LIN {X 0,Y 474.642,Z 379.86,A -85,B 0,C 180,E1 -7365.421,E2 -7365.421} C_VEL
LIN {X 0,Y 474.698,Z 379.855,A -85,B 0,C 180,E1 -7368.037,E2 -7368.037} C_VEL
LIN {X 0,Y 474.722,Z 379.85,A -85,B 0,C 180,E1 -7371.486,E2 -7371.486} C_VEL
LIN {X 0,Y 474.772,Z 379.846,A -85,B 0,C 180,E1 -7374.052,E2 -7374.052} C_VEL
LIN {X 0,Y 474.888,Z 379.83,A -85,B 0,C 180,E1 -7377.455,E2 -7377.455} C_VEL
LIN {X 0,Y 474.905,Z 379.83,A -85,B 0,C 180,E1 -7380,E2 -7380} C_VEL
LIN {X 0,Y 474.888,Z 379.832,A -85,B 0,C 180,E1 -7382.545,E2 -7382.545} C_VEL
LIN {X 0,Y 474.773,Z 379.846,A -85,B 0,C 180,E1 -7385.948,E2 -7385.948} C_VEL
LIN {X 0,Y 474.722,Z 379.853,A -85,B 0,C 180,E1 -7388.514,E2 -7388.514} C_VEL
LIN {X 0,Y 474.697,Z 379.856,A -85,B 0,C 180,E1 -7391.963,E2 -7391.963} C_VEL
LIN {X 0,Y 474.694,Z 379.855,A -85,B 0,C 180,E1 -7395.456,E2 -7395.456} C_VEL
LIN {X 0,Y 474.66,Z 379.858,A -85,B 0,C 180,E1 -7399.01,E2 -7399.01} C_VEL
LIN {X 0,Y 474.585,Z 379.871,A -85,B 0,C 180,E1 -7401.729,E2 -7401.729} C_VEL
LIN {X 0,Y 474.654,Z 379.86,A -85,B 0,C 180,E1 -7404.493,E2 -7404.493} C_VEL
LIN {X 0,Y 474.694,Z 379.855,A -85,B 0,C 180,E1 -7407.339,E2 -7407.339} C_VEL
LIN {X 0,Y 474.605,Z 379.865,A -85,B 0,C 180,E1 -7410.812,E2 -7410.812} C_VEL
LIN {X 0,Y 474.634,Z 379.862,A -85,B 0,C 180,E1 -7413.984,E2 -7413.984} C_VEL
LIN {X 0,Y 474.571,Z 379.869,A -85,B 0,C 180,E1 -7416.9,E2 -7416.9} C_VEL
LIN {X 0,Y 474.624,Z 379.865,A -85,B 0,C 180,E1 -7419.648,E2 -7419.648} C_VEL
LIN {X 0,Y 474.632,Z 379.862,A -85,B 0,C 180,E1 -7422.932,E2 -7422.932} C_VEL
LIN {X 0,Y 474.607,Z 379.865,A -85,B 0,C 180,E1 -7425.896,E2 -7425.896} C_VEL
LIN {X 0,Y 474.639,Z 379.862,A -85,B 0,C 180,E1 -7429.039,E2 -7429.039} C_VEL
LIN {X 0,Y 474.615,Z 379.864,A -85,B 0,C 180,E1 -7431.703,E2 -7431.703} C_VEL
LIN {X 0,Y 474.629,Z 379.861,A -85,B 0,C 180,E1 -7434.727,E2 -7434.727} C_VEL
LIN {X 0,Y 474.635,Z 379.861,A -85,B 0,C 180,E1 -7437.788,E2 -7437.788} C_VEL
LIN {X 0,Y 474.624,Z 379.864,A -85,B 0,C 180,E1 -7440.885,E2 -7440.885} C_VEL
LIN {X 0,Y 474.661,Z 379.858,A -85,B 0,C 180,E1 -7443.629,E2 -7443.629} C_VEL
LIN {X 0,Y 474.636,Z 379.861,A -85,B 0,C 180,E1 -7446.642,E2 -7446.642} C_VEL
LIN {X 0,Y 474.656,Z 379.856,A -85,B 0,C 180,E1 -7450.09,E2 -7450.09} C_VEL
LIN {X 0,Y 474.656,Z 379.857,A -85,B 0,C 180,E1 -7451.682,E2 -7451.682} C_VEL
LIN {X 0,Y 473.992,Z 379.94,A -85,B 0,C 180,E1 -7452.391,E2 -7452.391} C_VEL
LIN {X 0,Y 471.142,Z 380.3,A -85,B 0,C 180,E1 -7453.543,E2 -7453.543} C_VEL
LIN {X 0,Y 468.726,Z 380.603,A -85,B 0,C 180,E1 -7454.471,E2 -7454.471} C_VEL
LIN {X 0,Y 467.685,Z 380.731,A -85,B 0,C 180,E1 -7455.188,E2 -7455.188} C_VEL
LIN {X 0,Y 467.599,Z 380.739,A -85,B 0,C 180,E1 -7455.431,E2 -7455.431} C_VEL
LIN {X 0,Y 467.655,Z 380.734,A -85,B 0,C 180,E1 -7458.734,E2 -7458.734} C_VEL
LIN {X 0,Y 467.685,Z 380.853,A -85,B 0,C 180,E1 -7460.049,E2 -7460.049} C_VEL
LIN {X 0,Y 469.106,Z 388.705,A -85,B 0,C 180,E1 -7461.779,E2 -7461.779} C_VEL
LIN {X 0,Y 468.743,Z 398.423,A -85,B 0,C 180,E1 -7463.759,E2 -7463.759} C_VEL
LIN {X 0,Y 468.384,Z 409.921,A -85,B 0,C 180,E1 -7466.047,E2 -7466.047} C_VEL
LIN {X 0,Y 469.112,Z 414.147,A -85,B 0,C 180,E1 -7466.183,E2 -7466.183} C_VEL
LIN {X 0,Y 471.27,Z 426.346,A -85,B 0,C 180,E1 -7466.446,E2 -7466.446} C_VEL
LIN {X 0,Y 470.532,Z 517.39,A -85,B 0,C 180,E1 -7467.86,E2 -7467.86} C_VEL
LIN {X 0,Y 470.19,Z 531.181,A -85,B 0,C 180,E1 -7468.26,E2 -7468.26} C_VEL
LIN {X 0,Y 469.819,Z 544.038,A -85,B 0,C 180,E1 -7468.821,E2 -7468.821} C_VEL
LIN {X 0,Y 469.283,Z 556.55,A -85,B 0,C 180,E1 -7469.571,E2 -7469.571} C_VEL
LIN {X 0,Y 468.732,Z 567.702,A -85,B 0,C 180,E1 -7470.429,E2 -7470.429} C_VEL
LIN {X 0,Y 468.308,Z 576.724,A -85,B 0,C 180,E1 -7471.29,E2 -7471.29} C_VEL
LIN {X 0,Y 467.868,Z 586.01,A -85,B 0,C 180,E1 -7472.367,E2 -7472.367} C_VEL
LIN {X 0,Y 467.406,Z 595.008,A -85,B 0,C 180,E1 -7473.664,E2 -7473.664} C_VEL
LIN {X 0,Y 467.034,Z 602.282,A -85,B 0,C 180,E1 -7474.964,E2 -7474.964} C_VEL
LIN {X 0,Y 466.932,Z 608.355,A -85,B 0,C 180,E1 -7476.328,E2 -7476.328} C_VEL
LIN {X 0,Y 466.768,Z 613.344,A -85,B 0,C 180,E1 -7477.788,E2 -7477.788} C_VEL
LIN {X 0,Y 466.684,Z 615.684,A -85,B 0,C 180,E1 -7478.661,E2 -7478.661} C_VEL
LIN {X 0,Y 466.575,Z 617.597,A -85,B 0,C 180,E1 -7479.537,E2 -7479.537} C_VEL
LIN {X 0,Y 466.601,Z 619.039,A -85,B 0,C 180,E1 -7480.413,E2 -7480.413} C_VEL
LIN {X 0,Y 466.627,Z 620.462,A -85,B 0,C 180,E1 -7481.767,E2 -7481.767} C_VEL
LIN {X 0,Y 466.545,Z 620.916,A -85,B 0,C 180,E1 -7483.059,E2 -7483.059} C_VEL
LIN {X 0,Y 466.506,Z 620.687,A -85,B 0,C 180,E1 -7483.948,E2 -7483.948} C_VEL
LIN {X 0,Y 466.582,Z 619.413,A -85,B 0,C 180,E1 -7485.417,E2 -7485.417} C_VEL
LIN {X 0,Y 466.575,Z 617.498,A -85,B 0,C 180,E1 -7486.63,E2 -7486.63} C_VEL
LIN {X 0,Y 466.722,Z 614.362,A -85,B 0,C 180,E1 -7487.98,E2 -7487.98} C_VEL
LIN {X 0,Y 466.873,Z 610.064,A -85,B 0,C 180,E1 -7489.339,E2 -7489.339} C_VEL
LIN {X 0,Y 467.114,Z 603.53,A -85,B 0,C 180,E1 -7490.908,E2 -7490.908} C_VEL
LIN {X 0,Y 467.476,Z 596.001,A -85,B 0,C 180,E1 -7492.309,E2 -7492.309} C_VEL
LIN {X 0,Y 467.885,Z 587.185,A -85,B 0,C 180,E1 -7493.613,E2 -7493.613} C_VEL
LIN {X 0,Y 468.357,Z 577.917,A -85,B 0,C 180,E1 -7494.725,E2 -7494.725} C_VEL
LIN {X 0,Y 468.885,Z 567.133,A -85,B 0,C 180,E1 -7495.764,E2 -7495.764} C_VEL
LIN {X 0,Y 469.394,Z 556.525,A -85,B 0,C 180,E1 -7496.58,E2 -7496.58} C_VEL
LIN {X 0,Y 469.876,Z 545.344,A -85,B 0,C 180,E1 -7497.261,E2 -7497.261} C_VEL
LIN {X 0,Y 470.301,Z 533.471,A -85,B 0,C 180,E1 -7497.81,E2 -7497.81} C_VEL
LIN {X 0,Y 470.598,Z 520.548,A -85,B 0,C 180,E1 -7498.222,E2 -7498.222} C_VEL
LIN {X 0,Y 470.832,Z 503.541,A -85,B 0,C 180,E1 -7498.532,E2 -7498.532} C_VEL
LIN {X 0,Y 471.437,Z 425.884,A -85,B 0,C 180,E1 -7499.73,E2 -7499.73} C_VEL
LIN {X 0,Y 468.522,Z 410.206,A -85,B 0,C 180,E1 -7500.122,E2 -7500.122} C_VEL
LIN {X 0,Y 468.767,Z 404.216,A -85,B 0,C 180,E1 -7501.287,E2 -7501.287} C_VEL
LIN {X 0,Y 469.373,Z 391.54,A -85,B 0,C 180,E1 -7503.899,E2 -7503.899} C_VEL
LIN {X 0,Y 468.511,Z 385.277,A -85,B 0,C 180,E1 -7505.276,E2 -7505.276} C_VEL
LIN {X 0,Y 467.577,Z 380.785,A -85,B 0,C 180,E1 -7506.353,E2 -7506.353} C_VEL
LIN {X 0,Y 467.615,Z 380.739,A -85,B 0,C 180,E1 -7509.14,E2 -7509.14} C_VEL
LIN {X 0,Y 467.615,Z 380.737,A -85,B 0,C 180,E1 -7512.571,E2 -7512.571} C_VEL
LIN {X 0,Y 467.569,Z 380.74,A -85,B 0,C 180,E1 -7516.176,E2 -7516.176} C_VEL
LIN {X 0,Y 467.585,Z 380.737,A -85,B 0,C 180,E1 -7518.721,E2 -7518.721} C_VEL
LIN {X 0,Y 467.572,Z 380.739,A -85,B 0,C 180,E1 -7521.406,E2 -7521.406} C_VEL
LIN {X 0,Y 467.557,Z 380.74,A -85,B 0,C 180,E1 -7524.259,E2 -7524.259} C_VEL
LIN {X 0,Y 467.575,Z 380.743,A -85,B 0,C 180,E1 -7527.32,E2 -7527.32} C_VEL
LIN {X 0,Y 467.571,Z 380.732,A -85,B 0,C 180,E1 -7530.665,E2 -7530.665} C_VEL
LIN {X 0,Y 467.62,Z 380.738,A -85,B 0,C 180,E1 -7533.2,E2 -7533.2} C_VEL
LIN {X 0,Y 467.585,Z 380.739,A -85,B 0,C 180,E1 -7536.467,E2 -7536.467} C_VEL
LIN {X 0,Y 467.617,Z 380.733,A -85,B 0,C 180,E1 -7539.777,E2 -7539.777} C_VEL
LIN {X 0,Y 467.6,Z 380.735,A -85,B 0,C 180,E1 -7542.506,E2 -7542.506} C_VEL
LIN {X 0,Y 467.598,Z 380.736,A -85,B 0,C 180,E1 -7545.196,E2 -7545.196} C_VEL
LIN {X 0,Y 467.673,Z 380.726,A -85,B 0,C 180,E1 -7547.855,E2 -7547.855} C_VEL
LIN {X 0,Y 467.674,Z 380.728,A -85,B 0,C 180,E1 -7551.357,E2 -7551.357} C_VEL
LIN {X 0,Y 467.738,Z 380.714,A -85,B 0,C 180,E1 -7553.963,E2 -7553.963} C_VEL
LIN {X 0,Y 467.858,Z 380.703,A -85,B 0,C 180,E1 -7557.417,E2 -7557.417} C_VEL
LIN {X 0,Y 467.873,Z 380.698,A -85,B 0,C 180,E1 -7560,E2 -7560} C_VEL
LIN {X 0,Y 467.852,Z 380.709,A -85,B 0,C 180,E1 -7562.583,E2 -7562.583} C_VEL
LIN {X 0,Y 467.739,Z 380.718,A -85,B 0,C 180,E1 -7566.038,E2 -7566.038} C_VEL
LIN {X 0,Y 467.674,Z 380.727,A -85,B 0,C 180,E1 -7568.643,E2 -7568.643} C_VEL
LIN {X 0,Y 467.674,Z 380.727,A -85,B 0,C 180,E1 -7572.145,E2 -7572.145} C_VEL
LIN {X 0,Y 467.64,Z 380.73,A -85,B 0,C 180,E1 -7575.886,E2 -7575.886} C_VEL
LIN {X 0,Y 467.616,Z 380.733,A -85,B 0,C 180,E1 -7579.308,E2 -7579.308} C_VEL
LIN {X 0,Y 467.534,Z 380.743,A -85,B 0,C 180,E1 -7582.074,E2 -7582.074} C_VEL
LIN {X 0,Y 467.598,Z 380.739,A -85,B 0,C 180,E1 -7584.888,E2 -7584.888} C_VEL
LIN {X 0,Y 467.62,Z 380.731,A -85,B 0,C 180,E1 -7587.769,E2 -7587.769} C_VEL
LIN {X 0,Y 467.562,Z 380.742,A -85,B 0,C 180,E1 -7591.046,E2 -7591.046} C_VEL
LIN {X 0,Y 467.584,Z 380.739,A -85,B 0,C 180,E1 -7594.243,E2 -7594.243} C_VEL
LIN {X 0,Y 467.545,Z 380.741,A -85,B 0,C 180,E1 -7597.188,E2 -7597.188} C_VEL
LIN {X 0,Y 467.591,Z 380.74,A -85,B 0,C 180,E1 -7600.263,E2 -7600.263} C_VEL
LIN {X 0,Y 467.614,Z 380.732,A -85,B 0,C 180,E1 -7602.572,E2 -7602.572} C_VEL
LIN {X 0,Y 467.563,Z 380.739,A -85,B 0,C 180,E1 -7606.178,E2 -7606.178} C_VEL
LIN {X 0,Y 467.578,Z 380.741,A -85,B 0,C 180,E1 -7608.724,E2 -7608.724} C_VEL
LIN {X 0,Y 467.564,Z 380.743,A -85,B 0,C 180,E1 -7611.957,E2 -7611.957} C_VEL
LIN {X 0,Y 467.567,Z 380.74,A -85,B 0,C 180,E1 -7615.169,E2 -7615.169} C_VEL
LIN {X 0,Y 467.583,Z 380.741,A -85,B 0,C 180,E1 -7618.261,E2 -7618.261} C_VEL
LIN {X 0,Y 467.577,Z 380.741,A -85,B 0,C 180,E1 -7621.251,E2 -7621.251} C_VEL
LIN {X 0,Y 467.612,Z 380.739,A -85,B 0,C 180,E1 -7624.161,E2 -7624.161} C_VEL
LIN {X 0,Y 467.657,Z 380.901,A -85,B 0,C 180,E1 -7624.903,E2 -7624.903} C_VEL
LIN {X 0,Y 469.631,Z 391.304,A -85,B 0,C 180,E1 -7627.103,E2 -7627.103} C_VEL
LIN {X 0,Y 469.655,Z 396.068,A -85,B 0,C 180,E1 -7628.032,E2 -7628.032} C_VEL
LIN {X 0,Y 468.787,Z 414.077,A -85,B 0,C 180,E1 -7631.438,E2 -7631.438} C_VEL
LIN {X 0,Y 468.449,Z 422.17,A -85,B 0,C 180,E1 -7632.905,E2 -7632.905} C_VEL
LIN {X 0,Y 469.901,Z 430.791,A -85,B 0,C 180,E1 -7633.133,E2 -7633.133} C_VEL
LIN {X 0,Y 471.376,Z 440.03,A -85,B 0,C 180,E1 -7633.338,E2 -7633.338} C_VEL
LIN {X 0,Y 470.646,Z 529.828,A -85,B 0,C 180,E1 -7634.741,E2 -7634.741} C_VEL
LIN {X 0,Y 470.312,Z 543.065,A -85,B 0,C 180,E1 -7635.118,E2 -7635.118} C_VEL
LIN {X 0,Y 469.856,Z 555.767,A -85,B 0,C 180,E1 -7635.657,E2 -7635.657} C_VEL
LIN {X 0,Y 469.352,Z 567.861,A -85,B 0,C 180,E1 -7636.36,E2 -7636.36} C_VEL
LIN {X 0,Y 468.852,Z 578.48,A -85,B 0,C 180,E1 -7637.152,E2 -7637.152} C_VEL
LIN {X 0,Y 468.356,Z 589.73,A -85,B 0,C 180,E1 -7638.203,E2 -7638.203} C_VEL
LIN {X 0,Y 467.884,Z 598.212,A -85,B 0,C 180,E1 -7639.178,E2 -7639.178} C_VEL
LIN {X 0,Y 467.442,Z 607.416,A -85,B 0,C 180,E1 -7640.481,E2 -7640.481} C_VEL
LIN {X 0,Y 467.118,Z 614.819,A -85,B 0,C 180,E1 -7641.783,E2 -7641.783} C_VEL
LIN {X 0,Y 466.912,Z 620.766,A -85,B 0,C 180,E1 -7643.084,E2 -7643.084} C_VEL
LIN {X 0,Y 466.794,Z 625.466,A -85,B 0,C 180,E1 -7644.384,E2 -7644.384} C_VEL
LIN {X 0,Y 466.648,Z 629.056,A -85,B 0,C 180,E1 -7645.682,E2 -7645.682} C_VEL
LIN {X 0,Y 466.661,Z 630.908,A -85,B 0,C 180,E1 -7646.547,E2 -7646.547} C_VEL
LIN {X 0,Y 466.644,Z 632.297,A -85,B 0,C 180,E1 -7647.411,E2 -7647.411} C_VEL
LIN {X 0,Y 466.589,Z 633.893,A -85,B 0,C 180,E1 -7649.137,E2 -7649.137} C_VEL
LIN {X 0,Y 466.598,Z 634.105,A -85,B 0,C 180,E1 -7650,E2 -7650} C_VEL
LIN {X 0,Y 466.604,Z 633.278,A -85,B 0,C 180,E1 -7651.726,E2 -7651.726} C_VEL
LIN {X 0,Y 466.644,Z 632.283,A -85,B 0,C 180,E1 -7652.59,E2 -7652.59} C_VEL
LIN {X 0,Y 466.661,Z 630.885,A -85,B 0,C 180,E1 -7653.454,E2 -7653.454} C_VEL
LIN {X 0,Y 466.693,Z 627.949,A -85,B 0,C 180,E1 -7654.751,E2 -7654.751} C_VEL
LIN {X 0,Y 466.784,Z 623.972,A -85,B 0,C 180,E1 -7656.05,E2 -7656.05} C_VEL
LIN {X 0,Y 466.982,Z 617.847,A -85,B 0,C 180,E1 -7657.567,E2 -7657.567} C_VEL
LIN {X 0,Y 467.303,Z 611.156,A -85,B 0,C 180,E1 -7658.868,E2 -7658.868} C_VEL
LIN {X 0,Y 467.63,Z 602.848,A -85,B 0,C 180,E1 -7660.171,E2 -7660.171} C_VEL
LIN {X 0,Y 468.078,Z 594.311,A -85,B 0,C 180,E1 -7661.256,E2 -7661.256} C_VEL
LIN {X 0,Y 468.605,Z 583.971,A -85,B 0,C 180,E1 -7662.321,E2 -7662.321} C_VEL
LIN {X 0,Y 469.029,Z 573.591,A -85,B 0,C 180,E1 -7663.187,E2 -7663.187} C_VEL
LIN {X 0,Y 469.49,Z 561.79,A -85,B 0,C 180,E1 -7663.968,E2 -7663.968} C_VEL
LIN {X 0,Y 469.979,Z 549.854,A -85,B 0,C 180,E1 -7664.561,E2 -7664.561} C_VEL
LIN {X 0,Y 470.373,Z 536.957,A -85,B 0,C 180,E1 -7665.019,E2 -7665.019} C_VEL
LIN {X 0,Y 470.588,Z 523.354,A -85,B 0,C 180,E1 -7665.317,E2 -7665.317} C_VEL
LIN {X 0,Y 471.188,Z 439.488,A -85,B 0,C 180,E1 -7666.6,E2 -7666.6} C_VEL
LIN {X 0,Y 468.374,Z 422.324,A -85,B 0,C 180,E1 -7666.986,E2 -7666.986} C_VEL
LIN {X 0,Y 468.713,Z 413.473,A -85,B 0,C 180,E1 -7668.565,E2 -7668.565} C_VEL
LIN {X 0,Y 469.571,Z 393.96,A -85,B 0,C 180,E1 -7672.204,E2 -7672.204} C_VEL
LIN {X 0,Y 469.415,Z 390.298,A -85,B 0,C 180,E1 -7672.909,E2 -7672.909} C_VEL
LIN {X 0,Y 467.723,Z 381.106,A -85,B 0,C 180,E1 -7674.762,E2 -7674.762} C_VEL
LIN {X 0,Y 467.626,Z 380.739,A -85,B 0,C 180,E1 -7675.099,E2 -7675.099} C_VEL
LIN {X 0,Y 467.628,Z 380.736,A -85,B 0,C 180,E1 -7677.768,E2 -7677.768} C_VEL
LIN {X 0,Y 467.57,Z 380.743,A -85,B 0,C 180,E1 -7681.045,E2 -7681.045} C_VEL
LIN {X 0,Y 467.59,Z 380.737,A -85,B 0,C 180,E1 -7684.242,E2 -7684.242} C_VEL
LIN {X 0,Y 467.552,Z 380.745,A -85,B 0,C 180,E1 -7687.186,E2 -7687.186} C_VEL
LIN {X 0,Y 467.578,Z 380.738,A -85,B 0,C 180,E1 -7690.264,E2 -7690.264} C_VEL
LIN {X 0,Y 467.585,Z 380.738,A -85,B 0,C 180,E1 -7692.566,E2 -7692.566} C_VEL
LIN {X 0,Y 467.569,Z 380.743,A -85,B 0,C 180,E1 -7695.053,E2 -7695.053} C_VEL
LIN {X 0,Y 467.622,Z 380.738,A -85,B 0,C 180,E1 -7697.443,E2 -7697.443} C_VEL
LIN {X 0,Y 467.616,Z 380.736,A -85,B 0,C 180,E1 -7700.858,E2 -7700.858} C_VEL
LIN {X 0,Y 467.56,Z 380.742,A -85,B 0,C 180,E1 -7704.26,E2 -7704.26} C_VEL
LIN {X 0,Y 467.578,Z 380.743,A -85,B 0,C 180,E1 -7707.32,E2 -7707.32} C_VEL
LIN {X 0,Y 467.566,Z 380.742,A -85,B 0,C 180,E1 -7710.667,E2 -7710.667} C_VEL
LIN {X 0,Y 467.623,Z 380.738,A -85,B 0,C 180,E1 -7713.2,E2 -7713.2} C_VEL
LIN {X 0,Y 467.588,Z 380.74,A -85,B 0,C 180,E1 -7716.468,E2 -7716.468} C_VEL
LIN {X 0,Y 467.619,Z 380.735,A -85,B 0,C 180,E1 -7719.777,E2 -7719.777} C_VEL
LIN {X 0,Y 467.604,Z 380.738,A -85,B 0,C 180,E1 -7722.506,E2 -7722.506} C_VEL
LIN {X 0,Y 467.6,Z 380.739,A -85,B 0,C 180,E1 -7725.196,E2 -7725.196} C_VEL
LIN {X 0,Y 467.649,Z 380.732,A -85,B 0,C 180,E1 -7727.854,E2 -7727.854} C_VEL
LIN {X 0,Y 467.675,Z 380.728,A -85,B 0,C 180,E1 -7731.357,E2 -7731.357} C_VEL
LIN {X 0,Y 467.737,Z 380.722,A -85,B 0,C 180,E1 -7733.962,E2 -7733.962} C_VEL
LIN {X 0,Y 467.854,Z 380.706,A -85,B 0,C 180,E1 -7737.417,E2 -7737.417} C_VEL
LIN {X 0,Y 467.876,Z 380.705,A -85,B 0,C 180,E1 -7740,E2 -7740} C_VEL
LIN {X 0,Y 467.854,Z 380.708,A -85,B 0,C 180,E1 -7742.583,E2 -7742.583} C_VEL
LIN {X 0,Y 467.737,Z 380.722,A -85,B 0,C 180,E1 -7746.037,E2 -7746.037} C_VEL
LIN {X 0,Y 467.675,Z 380.731,A -85,B 0,C 180,E1 -7748.643,E2 -7748.643} C_VEL
LIN {X 0,Y 467.649,Z 380.733,A -85,B 0,C 180,E1 -7752.146,E2 -7752.146} C_VEL
LIN {X 0,Y 467.633,Z 380.737,A -85,B 0,C 180,E1 -7755.695,E2 -7755.695} C_VEL
LIN {X 0,Y 467.612,Z 380.737,A -85,B 0,C 180,E1 -7758.765,E2 -7758.765} C_VEL
LIN {X 0,Y 467.575,Z 380.741,A -85,B 0,C 180,E1 -7761.269,E2 -7761.269} C_VEL
LIN {X 0,Y 467.568,Z 380.743,A -85,B 0,C 180,E1 -7763.944,E2 -7763.944} C_VEL
LIN {X 0,Y 467.622,Z 380.735,A -85,B 0,C 180,E1 -7766.8,E2 -7766.8} C_VEL
LIN {X 0,Y 467.583,Z 380.742,A -85,B 0,C 180,E1 -7769.736,E2 -7769.736} C_VEL
LIN {X 0,Y 467.579,Z 380.74,A -85,B 0,C 180,E1 -7772.759,E2 -7772.759} C_VEL
LIN {X 0,Y 467.553,Z 380.744,A -85,B 0,C 180,E1 -7775.89,E2 -7775.89} C_VEL
LIN {X 0,Y 467.579,Z 380.742,A -85,B 0,C 180,E1 -7779.145,E2 -7779.145} C_VEL
LIN {X 0,Y 467.583,Z 380.739,A -85,B 0,C 180,E1 -7782.567,E2 -7782.567} C_VEL
LIN {X 0,Y 467.568,Z 380.743,A -85,B 0,C 180,E1 -7785.054,E2 -7785.054} C_VEL
LIN {X 0,Y 467.586,Z 380.742,A -85,B 0,C 180,E1 -7787.44,E2 -7787.44} C_VEL
LIN {X 0,Y 467.614,Z 380.736,A -85,B 0,C 180,E1 -7790.859,E2 -7790.859} C_VEL
LIN {X 0,Y 467.562,Z 380.741,A -85,B 0,C 180,E1 -7794.261,E2 -7794.261} C_VEL
LIN {X 0,Y 467.581,Z 380.743,A -85,B 0,C 180,E1 -7797.321,E2 -7797.321} C_VEL
LIN {X 0,Y 467.57,Z 380.741,A -85,B 0,C 180,E1 -7800.668,E2 -7800.668} C_VEL
LIN {X 0,Y 467.617,Z 380.739,A -85,B 0,C 180,E1 -7803.2,E2 -7803.2} C_VEL
LIN {X 0,Y 467.593,Z 380.737,A -85,B 0,C 180,E1 -7806.469,E2 -7806.469} C_VEL
LIN {X 0,Y 467.624,Z 380.733,A -85,B 0,C 180,E1 -7809.777,E2 -7809.777} C_VEL
LIN {X 0,Y 467.608,Z 380.736,A -85,B 0,C 180,E1 -7812.507,E2 -7812.507} C_VEL
LIN {X 0,Y 467.599,Z 380.739,A -85,B 0,C 180,E1 -7815.431,E2 -7815.431} C_VEL
LIN {X 0,Y 466.928,Z 380.82,A -85,B 0,C 180,E1 -7816.15,E2 -7816.15} C_VEL
LIN {X 0,Y 464.085,Z 381.178,A -85,B 0,C 180,E1 -7817.319,E2 -7817.319} C_VEL
LIN {X 0,Y 461.686,Z 381.476,A -85,B 0,C 180,E1 -7818.261,E2 -7818.261} C_VEL
LIN {X 0,Y 460.66,Z 381.605,A -85,B 0,C 180,E1 -7818.988,E2 -7818.988} C_VEL
LIN {X 0,Y 460.579,Z 381.614,A -85,B 0,C 180,E1 -7819.235,E2 -7819.235} C_VEL
LIN {X 0,Y 460.657,Z 381.768,A -85,B 0,C 180,E1 -7819.895,E2 -7819.895} C_VEL
LIN {X 0,Y 462.108,Z 389.84,A -85,B 0,C 180,E1 -7821.691,E2 -7821.691} C_VEL
LIN {X 0,Y 461.936,Z 398.299,A -85,B 0,C 180,E1 -7823.448,E2 -7823.448} C_VEL
LIN {X 0,Y 461.698,Z 401.507,A -85,B 0,C 180,E1 -7824.102,E2 -7824.102} C_VEL
LIN {X 0,Y 461.395,Z 409.977,A -85,B 0,C 180,E1 -7825.796,E2 -7825.796} C_VEL
LIN {X 0,Y 461.901,Z 412.882,A -85,B 0,C 180,E1 -7825.91,E2 -7825.91} C_VEL
LIN {X 0,Y 464.4,Z 425.885,A -85,B 0,C 180,E1 -7826.204,E2 -7826.204} C_VEL
LIN {X 0,Y 463.665,Z 517.07,A -85,B 0,C 180,E1 -7827.638,E2 -7827.638} C_VEL
LIN {X 0,Y 463.326,Z 530.256,A -85,B 0,C 180,E1 -7828.017,E2 -7828.017} C_VEL
LIN {X 0,Y 462.916,Z 543.441,A -85,B 0,C 180,E1 -7828.586,E2 -7828.586} C_VEL
LIN {X 0,Y 462.456,Z 554.555,A -85,B 0,C 180,E1 -7829.238,E2 -7829.238} C_VEL
LIN {X 0,Y 461.879,Z 566.094,A -85,B 0,C 180,E1 -7830.109,E2 -7830.109} C_VEL
LIN {X 0,Y 461.329,Z 576.484,A -85,B 0,C 180,E1 -7831.091,E2 -7831.091} C_VEL
LIN {X 0,Y 460.871,Z 585.849,A -85,B 0,C 180,E1 -7832.185,E2 -7832.185} C_VEL
LIN {X 0,Y 460.373,Z 594.9,A -85,B 0,C 180,E1 -7833.501,E2 -7833.501} C_VEL
LIN {X 0,Y 459.994,Z 602.211,A -85,B 0,C 180,E1 -7834.82,E2 -7834.82} C_VEL
LIN {X 0,Y 459.89,Z 608.063,A -85,B 0,C 180,E1 -7836.141,E2 -7836.141} C_VEL
LIN {X 0,Y 459.697,Z 612.705,A -85,B 0,C 180,E1 -7837.466,E2 -7837.466} C_VEL
LIN {X 0,Y 459.565,Z 616.245,A -85,B 0,C 180,E1 -7838.796,E2 -7838.796} C_VEL
LIN {X 0,Y 459.475,Z 618.035,A -85,B 0,C 180,E1 -7839.686,E2 -7839.686} C_VEL
LIN {X 0,Y 459.497,Z 619.384,A -85,B 0,C 180,E1 -7840.576,E2 -7840.576} C_VEL
LIN {X 0,Y 459.546,Z 620.598,A -85,B 0,C 180,E1 -7841.826,E2 -7841.826} C_VEL
LIN {X 0,Y 459.428,Z 620.987,A -85,B 0,C 180,E1 -7843.265,E2 -7843.265} C_VEL
LIN {X 0,Y 459.43,Z 620.682,A -85,B 0,C 180,E1 -7844.167,E2 -7844.167} C_VEL
LIN {X 0,Y 459.493,Z 619.461,A -85,B 0,C 180,E1 -7845.508,E2 -7845.508} C_VEL
LIN {X 0,Y 459.558,Z 616.248,A -85,B 0,C 180,E1 -7847.35,E2 -7847.35} C_VEL
LIN {X 0,Y 459.728,Z 612.577,A -85,B 0,C 180,E1 -7848.725,E2 -7848.725} C_VEL
LIN {X 0,Y 459.895,Z 607.676,A -85,B 0,C 180,E1 -7850.11,E2 -7850.11} C_VEL
LIN {X 0,Y 460.171,Z 601.386,A -85,B 0,C 180,E1 -7851.502,E2 -7851.502} C_VEL
LIN {X 0,Y 460.594,Z 593.467,A -85,B 0,C 180,E1 -7852.897,E2 -7852.897} C_VEL
LIN {X 0,Y 461.085,Z 584.547,A -85,B 0,C 180,E1 -7854.149,E2 -7854.149} C_VEL
LIN {X 0,Y 461.536,Z 575.027,A -85,B 0,C 180,E1 -7855.236,E2 -7855.236} C_VEL
LIN {X 0,Y 462.166,Z 563.828,A -85,B 0,C 180,E1 -7856.265,E2 -7856.265} C_VEL
LIN {X 0,Y 462.664,Z 552.064,A -85,B 0,C 180,E1 -7857.11,E2 -7857.11} C_VEL
LIN {X 0,Y 463.289,Z 539.303,A -85,B 0,C 180,E1 -7857.805,E2 -7857.805} C_VEL
LIN {X 0,Y 463.668,Z 526.393,A -85,B 0,C 180,E1 -7858.306,E2 -7858.306} C_VEL
LIN {X 0,Y 463.927,Z 512.622,A -85,B 0,C 180,E1 -7858.641,E2 -7858.641} C_VEL
LIN {X 0,Y 464.605,Z 426.038,A -85,B 0,C 180,E1 -7860.009,E2 -7860.009} C_VEL
LIN {X 0,Y 461.61,Z 410.294,A -85,B 0,C 180,E1 -7860.419,E2 -7860.419} C_VEL
LIN {X 0,Y 461.732,Z 406.389,A -85,B 0,C 180,E1 -7861.165,E2 -7861.165} C_VEL
LIN {X 0,Y 462.432,Z 393.06,A -85,B 0,C 180,E1 -7863.952,E2 -7863.952} C_VEL
LIN {X 0,Y 461.896,Z 388.331,A -85,B 0,C 180,E1 -7865.001,E2 -7865.001} C_VEL
LIN {X 0,Y 460.519,Z 381.649,A -85,B 0,C 180,E1 -7866.609,E2 -7866.609} C_VEL
LIN {X 0,Y 460.575,Z 381.615,A -85,B 0,C 180,E1 -7869.857,E2 -7869.857} C_VEL
LIN {X 0,Y 460.538,Z 381.618,A -85,B 0,C 180,E1 -7872.904,E2 -7872.904} C_VEL
LIN {X 0,Y 460.519,Z 381.619,A -85,B 0,C 180,E1 -7875.828,E2 -7875.828} C_VEL
LIN {X 0,Y 460.538,Z 381.618,A -85,B 0,C 180,E1 -7878.989,E2 -7878.989} C_VEL
LIN {X 0,Y 460.541,Z 381.614,A -85,B 0,C 180,E1 -7881.268,E2 -7881.268} C_VEL
LIN {X 0,Y 460.507,Z 381.62,A -85,B 0,C 180,E1 -7884.554,E2 -7884.554} C_VEL
LIN {X 0,Y 460.526,Z 381.618,A -85,B 0,C 180,E1 -7887.715,E2 -7887.715} C_VEL
LIN {X 0,Y 460.54,Z 381.609,A -85,B 0,C 180,E1 -7890.769,E2 -7890.769} C_VEL
LIN {X 0,Y 460.56,Z 381.612,A -85,B 0,C 180,E1 -7893.735,E2 -7893.735} C_VEL
LIN {X 0,Y 460.539,Z 381.619,A -85,B 0,C 180,E1 -7896.624,E2 -7896.624} C_VEL
LIN {X 0,Y 460.563,Z 381.614,A -85,B 0,C 180,E1 -7899.453,E2 -7899.453} C_VEL
LIN {X 0,Y 460.55,Z 381.611,A -85,B 0,C 180,E1 -7902.23,E2 -7902.23} C_VEL
LIN {X 0,Y 460.556,Z 381.615,A -85,B 0,C 180,E1 -7904.965,E2 -7904.965} C_VEL
LIN {X 0,Y 460.619,Z 381.605,A -85,B 0,C 180,E1 -7907.666,E2 -7907.666} C_VEL
LIN {X 0,Y 460.621,Z 381.608,A -85,B 0,C 180,E1 -7911.224,E2 -7911.224} C_VEL
LIN {X 0,Y 460.704,Z 381.59,A -85,B 0,C 180,E1 -7913.87,E2 -7913.87} C_VEL
LIN {X 0,Y 460.824,Z 381.579,A -85,B 0,C 180,E1 -7917.378,E2 -7917.378} C_VEL
LIN {X 0,Y 460.844,Z 381.574,A -85,B 0,C 180,E1 -7920,E2 -7920} C_VEL
LIN {X 0,Y 460.817,Z 381.585,A -85,B 0,C 180,E1 -7922.622,E2 -7922.622} C_VEL
LIN {X 0,Y 460.704,Z 381.594,A -85,B 0,C 180,E1 -7926.13,E2 -7926.13} C_VEL
LIN {X 0,Y 460.621,Z 381.605,A -85,B 0,C 180,E1 -7928.776,E2 -7928.776} C_VEL
LIN {X 0,Y 460.625,Z 381.608,A -85,B 0,C 180,E1 -7932.457,E2 -7932.457} C_VEL
LIN {X 0,Y 460.591,Z 381.609,A -85,B 0,C 180,E1 -7935.998,E2 -7935.998} C_VEL
LIN {X 0,Y 460.562,Z 381.615,A -85,B 0,C 180,E1 -7938.902,E2 -7938.902} C_VEL
LIN {X 0,Y 460.51,Z 381.617,A -85,B 0,C 180,E1 -7941.486,E2 -7941.486} C_VEL
LIN {X 0,Y 460.536,Z 381.617,A -85,B 0,C 180,E1 -7944.333,E2 -7944.333} C_VEL
LIN {X 0,Y 460.576,Z 381.61,A -85,B 0,C 180,E1 -7947.244,E2 -7947.244} C_VEL
LIN {X 0,Y 460.504,Z 381.621,A -85,B 0,C 180,E1 -7950.241,E2 -7950.241} C_VEL
LIN {X 0,Y 460.523,Z 381.616,A -85,B 0,C 180,E1 -7953.326,E2 -7953.326} C_VEL
LIN {X 0,Y 460.473,Z 381.629,A -85,B 0,C 180,E1 -7956.53,E2 -7956.53} C_VEL
LIN {X 0,Y 460.571,Z 381.611,A -85,B 0,C 180,E1 -7959.859,E2 -7959.859} C_VEL
LIN {X 0,Y 460.539,Z 381.618,A -85,B 0,C 180,E1 -7962.905,E2 -7962.905} C_VEL
LIN {X 0,Y 460.515,Z 381.615,A -85,B 0,C 180,E1 -7965.83,E2 -7965.83} C_VEL
LIN {X 0,Y 460.53,Z 381.616,A -85,B 0,C 180,E1 -7968.99,E2 -7968.99} C_VEL
LIN {X 0,Y 460.524,Z 381.618,A -85,B 0,C 180,E1 -7971.268,E2 -7971.268} C_VEL
LIN {X 0,Y 460.512,Z 381.624,A -85,B 0,C 180,E1 -7974.556,E2 -7974.556} C_VEL
LIN {X 0,Y 460.531,Z 381.618,A -85,B 0,C 180,E1 -7977.717,E2 -7977.717} C_VEL
LIN {X 0,Y 460.54,Z 381.621,A -85,B 0,C 180,E1 -7980.77,E2 -7980.77} C_VEL
LIN {X 0,Y 460.568,Z 381.617,A -85,B 0,C 180,E1 -7983.736,E2 -7983.736} C_VEL
LIN {X 0,Y 460.632,Z 381.838,A -85,B 0,C 180,E1 -7984.67,E2 -7984.67} C_VEL
LIN {X 0,Y 462.686,Z 392.573,A -85,B 0,C 180,E1 -7986.976,E2 -7986.976} C_VEL
LIN {X 0,Y 462.739,Z 397.174,A -85,B 0,C 180,E1 -7987.89,E2 -7987.89} C_VEL
LIN {X 0,Y 461.8,Z 415.227,A -85,B 0,C 180,E1 -7991.362,E2 -7991.362} C_VEL
LIN {X 0,Y 461.486,Z 421.95,A -85,B 0,C 180,E1 -7992.607,E2 -7992.607} C_VEL
LIN {X 0,Y 462.785,Z 429.059,A -85,B 0,C 180,E1 -7992.811,E2 -7992.811} C_VEL
LIN {X 0,Y 464.656,Z 441.523,A -85,B 0,C 180,E1 -7993.09,E2 -7993.09} C_VEL
LIN {X 0,Y 463.833,Z 530.506,A -85,B 0,C 180,E1 -7994.512,E2 -7994.512} C_VEL
LIN {X 0,Y 463.426,Z 544.235,A -85,B 0,C 180,E1 -7994.92,E2 -7994.92} C_VEL
LIN {X 0,Y 462.958,Z 557.078,A -85,B 0,C 180,E1 -7995.495,E2 -7995.495} C_VEL
LIN {X 0,Y 462.452,Z 568.322,A -85,B 0,C 180,E1 -7996.174,E2 -7996.174} C_VEL
LIN {X 0,Y 461.88,Z 579.389,A -85,B 0,C 180,E1 -7997.025,E2 -7997.025} C_VEL
LIN {X 0,Y 461.396,Z 589.784,A -85,B 0,C 180,E1 -7998.022,E2 -7998.022} C_VEL
LIN {X 0,Y 460.896,Z 598.234,A -85,B 0,C 180,E1 -7999.012,E2 -7999.012} C_VEL
LIN {X 0,Y 460.412,Z 607.403,A -85,B 0,C 180,E1 -8000.334,E2 -8000.334} C_VEL
LIN {X 0,Y 460.077,Z 614.787,A -85,B 0,C 180,E1 -8001.656,E2 -8001.656} C_VEL
LIN {X 0,Y 459.846,Z 620.718,A -85,B 0,C 180,E1 -8002.977,E2 -8002.977} C_VEL
LIN {X 0,Y 459.712,Z 625.405,A -85,B 0,C 180,E1 -8004.297,E2 -8004.297} C_VEL
LIN {X 0,Y 459.566,Z 628.984,A -85,B 0,C 180,E1 -8005.615,E2 -8005.615} C_VEL
LIN {X 0,Y 459.558,Z 630.828,A -85,B 0,C 180,E1 -8006.493,E2 -8006.493} C_VEL
LIN {X 0,Y 459.566,Z 632.21,A -85,B 0,C 180,E1 -8007.371,E2 -8007.371} C_VEL
LIN {X 0,Y 459.494,Z 633.798,A -85,B 0,C 180,E1 -8009.124,E2 -8009.124} C_VEL
LIN {X 0,Y 459.501,Z 634.004,A -85,B 0,C 180,E1 -8010,E2 -8010} C_VEL
LIN {X 0,Y 459.516,Z 633.167,A -85,B 0,C 180,E1 -8011.753,E2 -8011.753} C_VEL
LIN {X 0,Y 459.566,Z 632.169,A -85,B 0,C 180,E1 -8012.63,E2 -8012.63} C_VEL
LIN {X 0,Y 459.558,Z 630.763,A -85,B 0,C 180,E1 -8013.507,E2 -8013.507} C_VEL
LIN {X 0,Y 459.625,Z 627.819,A -85,B 0,C 180,E1 -8014.824,E2 -8014.824} C_VEL
LIN {X 0,Y 459.717,Z 622.777,A -85,B 0,C 180,E1 -8016.434,E2 -8016.434} C_VEL
LIN {X 0,Y 459.965,Z 616.674,A -85,B 0,C 180,E1 -8017.904,E2 -8017.904} C_VEL
LIN {X 0,Y 460.28,Z 609.737,A -85,B 0,C 180,E1 -8019.226,E2 -8019.226} C_VEL
LIN {X 0,Y 460.67,Z 601.033,A -85,B 0,C 180,E1 -8020.549,E2 -8020.549} C_VEL
LIN {X 0,Y 461.185,Z 592.113,A -85,B 0,C 180,E1 -8021.649,E2 -8021.649} C_VEL
LIN {X 0,Y 461.71,Z 581.991,A -85,B 0,C 180,E1 -8022.669,E2 -8022.669} C_VEL
LIN {X 0,Y 462.208,Z 571.526,A -85,B 0,C 180,E1 -8023.52,E2 -8023.52} C_VEL
LIN {X 0,Y 462.662,Z 559.396,A -85,B 0,C 180,E1 -8024.291,E2 -8024.291} C_VEL
LIN {X 0,Y 463.175,Z 546.729,A -85,B 0,C 180,E1 -8024.892,E2 -8024.892} C_VEL
LIN {X 0,Y 463.562,Z 534.325,A -85,B 0,C 180,E1 -8025.301,E2 -8025.301} C_VEL
LIN {X 0,Y 463.733,Z 518.506,A -85,B 0,C 180,E1 -8025.605,E2 -8025.605} C_VEL
LIN {X 0,Y 464.355,Z 440.838,A -85,B 0,C 180,E1 -8026.809,E2 -8026.809} C_VEL
LIN {X 0,Y 461.398,Z 422.39,A -85,B 0,C 180,E1 -8027.217,E2 -8027.217} C_VEL
LIN {X 0,Y 461.468,Z 419.25,A -85,B 0,C 180,E1 -8027.734,E2 -8027.734} C_VEL
LIN {X 0,Y 462.163,Z 403.467,A -85,B 0,C 180,E1 -8030.705,E2 -8030.705} C_VEL
LIN {X 0,Y 462.6,Z 392.498,A -85,B 0,C 180,E1 -8032.793,E2 -8032.793} C_VEL
LIN {X 0,Y 460.625,Z 381.825,A -85,B 0,C 180,E1 -8034.989,E2 -8034.989} C_VEL
LIN {X 0,Y 460.557,Z 381.616,A -85,B 0,C 180,E1 -8038.232,E2 -8038.232} C_VEL
LIN {X 0,Y 460.523,Z 381.623,A -85,B 0,C 180,E1 -8041.283,E2 -8041.283} C_VEL
LIN {X 0,Y 460.534,Z 381.616,A -85,B 0,C 180,E1 -8044.505,E2 -8044.505} C_VEL
LIN {X 0,Y 460.529,Z 381.621,A -85,B 0,C 180,E1 -8047.62,E2 -8047.62} C_VEL
LIN {X 0,Y 460.542,Z 381.615,A -85,B 0,C 180,E1 -8050.269,E2 -8050.269} C_VEL
LIN {X 0,Y 460.508,Z 381.626,A -85,B 0,C 180,E1 -8053.374,E2 -8053.374} C_VEL
LIN {X 0,Y 460.523,Z 381.618,A -85,B 0,C 180,E1 -8056.627,E2 -8056.627} C_VEL
LIN {X 0,Y 460.558,Z 381.615,A -85,B 0,C 180,E1 -8059.727,E2 -8059.727} C_VEL
LIN {X 0,Y 460.526,Z 381.618,A -85,B 0,C 180,E1 -8062.518,E2 -8062.518} C_VEL
LIN {X 0,Y 460.545,Z 381.617,A -85,B 0,C 180,E1 -8065.623,E2 -8065.623} C_VEL
LIN {X 0,Y 460.533,Z 381.618,A -85,B 0,C 180,E1 -8068.744,E2 -8068.744} C_VEL
LIN {X 0,Y 460.584,Z 381.612,A -85,B 0,C 180,E1 -8072.252,E2 -8072.252} C_VEL
LIN {X 0,Y 460.555,Z 381.616,A -85,B 0,C 180,E1 -8074.705,E2 -8074.705} C_VEL
LIN {X 0,Y 460.506,Z 381.621,A -85,B 0,C 180,E1 -8077.571,E2 -8077.571} C_VEL
LIN {X 0,Y 460.564,Z 381.614,A -85,B 0,C 180,E1 -8080.384,E2 -8080.384} C_VEL
LIN {X 0,Y 460.56,Z 381.617,A -85,B 0,C 180,E1 -8083.146,E2 -8083.146} C_VEL
LIN {X 0,Y 460.548,Z 381.616,A -85,B 0,C 180,E1 -8085.868,E2 -8085.868} C_VEL
LIN {X 0,Y 460.605,Z 381.61,A -85,B 0,C 180,E1 -8088.559,E2 -8088.559} C_VEL
LIN {X 0,Y 460.689,Z 381.6,A -85,B 0,C 180,E1 -8092.108,E2 -8092.108} C_VEL
LIN {X 0,Y 460.691,Z 381.601,A -85,B 0,C 180,E1 -8094.748,E2 -8094.748} C_VEL
LIN {X 0,Y 460.819,Z 381.583,A -85,B 0,C 180,E1 -8097.378,E2 -8097.378} C_VEL
LIN {X 0,Y 460.846,Z 381.58,A -85,B 0,C 180,E1 -8100,E2 -8100} C_VEL
LIN {X 0,Y 460.819,Z 381.584,A -85,B 0,C 180,E1 -8102.622,E2 -8102.622} C_VEL
LIN {X 0,Y 460.704,Z 381.598,A -85,B 0,C 180,E1 -8106.13,E2 -8106.13} C_VEL
LIN {X 0,Y 460.622,Z 381.609,A -85,B 0,C 180,E1 -8108.776,E2 -8108.776} C_VEL
LIN {X 0,Y 460.607,Z 381.61,A -85,B 0,C 180,E1 -8112.445,E2 -8112.445} C_VEL
LIN {X 0,Y 460.594,Z 381.612,A -85,B 0,C 180,E1 -8115.998,E2 -8115.998} C_VEL
LIN {X 0,Y 460.565,Z 381.614,A -85,B 0,C 180,E1 -8118.902,E2 -8118.902} C_VEL
LIN {X 0,Y 460.51,Z 381.623,A -85,B 0,C 180,E1 -8121.486,E2 -8121.486} C_VEL
LIN {X 0,Y 460.537,Z 381.618,A -85,B 0,C 180,E1 -8124.333,E2 -8124.333} C_VEL
LIN {X 0,Y 460.579,Z 381.613,A -85,B 0,C 180,E1 -8127.243,E2 -8127.243} C_VEL
LIN {X 0,Y 460.523,Z 381.62,A -85,B 0,C 180,E1 -8130.239,E2 -8130.239} C_VEL
LIN {X 0,Y 460.525,Z 381.621,A -85,B 0,C 180,E1 -8133.325,E2 -8133.325} C_VEL
LIN {X 0,Y 460.475,Z 381.625,A -85,B 0,C 180,E1 -8136.53,E2 -8136.53} C_VEL
LIN {X 0,Y 460.541,Z 381.617,A -85,B 0,C 180,E1 -8138.898,E2 -8138.898} C_VEL
LIN {X 0,Y 460.521,Z 381.62,A -85,B 0,C 180,E1 -8142.182,E2 -8142.182} C_VEL
LIN {X 0,Y 460.514,Z 381.624,A -85,B 0,C 180,E1 -8145.412,E2 -8145.412} C_VEL
LIN {X 0,Y 460.533,Z 381.617,A -85,B 0,C 180,E1 -8148.397,E2 -8148.397} C_VEL
LIN {X 0,Y 460.543,Z 381.621,A -85,B 0,C 180,E1 -8151.269,E2 -8151.269} C_VEL
LIN {X 0,Y 460.513,Z 381.619,A -85,B 0,C 180,E1 -8154.555,E2 -8154.555} C_VEL
LIN {X 0,Y 460.531,Z 381.618,A -85,B 0,C 180,E1 -8157.716,E2 -8157.716} C_VEL
LIN {X 0,Y 460.54,Z 381.617,A -85,B 0,C 180,E1 -8160.769,E2 -8160.769} C_VEL
LIN {X 0,Y 460.563,Z 381.613,A -85,B 0,C 180,E1 -8163.735,E2 -8163.735} C_VEL
LIN {X 0,Y 460.546,Z 381.616,A -85,B 0,C 180,E1 -8166.624,E2 -8166.624} C_VEL
LIN {X 0,Y 460.552,Z 381.616,A -85,B 0,C 180,E1 -8169.453,E2 -8169.453} C_VEL
LIN {X 0,Y 460.559,Z 381.612,A -85,B 0,C 180,E1 -8172.23,E2 -8172.23} C_VEL
LIN {X 0,Y 460.567,Z 381.618,A -85,B 0,C 180,E1 -8174.965,E2 -8174.965} C_VEL
LIN {X 0,Y 460.613,Z 381.611,A -85,B 0,C 180,E1 -8178.559,E2 -8178.559} C_VEL
LIN {X 0,Y 460.579,Z 381.614,A -85,B 0,C 180,E1 -8179.235,E2 -8179.235} C_VEL
LIN {X 0,Y 460.344,Z 382.173,A -85,B 0,C 180,E1 -8179.719,E2 -8179.719} C_VEL
LIN {X 0,Y 459.756,Z 383.563,A -85,B 0,C 180,E1 -8180.177,E2 -8180.177} C_VEL
LIN {X 0,Y 457.978,Z 387.62,A -85,B 0,C 180,E1 -8181.028,E2 -8181.028} C_VEL
LIN {X 0,Y 455.374,Z 394.053,A -85,B 0,C 180,E1 -8182.268,E2 -8182.268} C_VEL
LIN {X 0,Y 454.983,Z 396.157,A -85,B 0,C 180,E1 -8182.696,E2 -8182.696} C_VEL
LIN {X 0,Y 454.747,Z 400.33,A -85,B 0,C 180,E1 -8183.567,E2 -8183.567} C_VEL
LIN {X 0,Y 454.483,Z 410.159,A -85,B 0,C 180,E1 -8185.565,E2 -8185.565} C_VEL
LIN {X 0,Y 455.12,Z 414.108,A -85,B 0,C 180,E1 -8185.695,E2 -8185.695} C_VEL
LIN {X 0,Y 457.55,Z 426.856,A -85,B 0,C 180,E1 -8185.981,E2 -8185.981} C_VEL
LIN {X 0,Y 456.783,Z 517.739,A -85,B 0,C 180,E1 -8187.437,E2 -8187.437} C_VEL
LIN {X 0,Y 456.41,Z 531.495,A -85,B 0,C 180,E1 -8187.849,E2 -8187.849} C_VEL
LIN {X 0,Y 456.002,Z 543.823,A -85,B 0,C 180,E1 -8188.399,E2 -8188.399} C_VEL
LIN {X 0,Y 455.472,Z 555.656,A -85,B 0,C 180,E1 -8189.116,E2 -8189.116} C_VEL
LIN {X 0,Y 454.902,Z 567.009,A -85,B 0,C 180,E1 -8190,E2 -8190} C_VEL
LIN {X 0,Y 454.304,Z 577.269,A -85,B 0,C 180,E1 -8190.997,E2 -8190.997} C_VEL
LIN {X 0,Y 453.872,Z 585.653,A -85,B 0,C 180,E1 -8191.996,E2 -8191.996} C_VEL
LIN {X 0,Y 453.351,Z 594.768,A -85,B 0,C 180,E1 -8193.332,E2 -8193.332} C_VEL
LIN {X 0,Y 452.964,Z 602.12,A -85,B 0,C 180,E1 -8194.672,E2 -8194.672} C_VEL
LIN {X 0,Y 452.78,Z 608.875,A -85,B 0,C 180,E1 -8196.237,E2 -8196.237} C_VEL
LIN {X 0,Y 452.619,Z 613.349,A -85,B 0,C 180,E1 -8197.584,E2 -8197.584} C_VEL
LIN {X 0,Y 452.463,Z 616.752,A -85,B 0,C 180,E1 -8198.935,E2 -8198.935} C_VEL
LIN {X 0,Y 452.384,Z 618.443,A -85,B 0,C 180,E1 -8199.839,E2 -8199.839} C_VEL
LIN {X 0,Y 452.399,Z 619.724,A -85,B 0,C 180,E1 -8200.743,E2 -8200.743} C_VEL
LIN {X 0,Y 452.445,Z 620.726,A -85,B 0,C 180,E1 -8201.873,E2 -8201.873} C_VEL
LIN {X 0,Y 452.34,Z 621.054,A -85,B 0,C 180,E1 -8203.476,E2 -8203.476} C_VEL
LIN {X 0,Y 452.341,Z 620.68,A -85,B 0,C 180,E1 -8204.394,E2 -8204.394} C_VEL
LIN {X 0,Y 452.395,Z 619.519,A -85,B 0,C 180,E1 -8205.597,E2 -8205.597} C_VEL
LIN {X 0,Y 452.439,Z 616.917,A -85,B 0,C 180,E1 -8207.165,E2 -8207.165} C_VEL
LIN {X 0,Y 452.634,Z 613.048,A -85,B 0,C 180,E1 -8208.712,E2 -8208.712} C_VEL
LIN {X 0,Y 452.807,Z 608.843,A -85,B 0,C 180,E1 -8209.965,E2 -8209.965} C_VEL
LIN {X 0,Y 453.108,Z 602.42,A -85,B 0,C 180,E1 -8211.465,E2 -8211.465} C_VEL
LIN {X 0,Y 453.493,Z 595.236,A -85,B 0,C 180,E1 -8212.794,E2 -8212.794} C_VEL
LIN {X 0,Y 453.97,Z 587.077,A -85,B 0,C 180,E1 -8214.022,E2 -8214.022} C_VEL
LIN {X 0,Y 454.469,Z 577.772,A -85,B 0,C 180,E1 -8215.167,E2 -8215.167} C_VEL
LIN {X 0,Y 455.084,Z 567.333,A -85,B 0,C 180,E1 -8216.197,E2 -8216.197} C_VEL
LIN {X 0,Y 455.679,Z 556.376,A -85,B 0,C 180,E1 -8217.063,E2 -8217.063} C_VEL
LIN {X 0,Y 456.217,Z 544.939,A -85,B 0,C 180,E1 -8217.774,E2 -8217.774} C_VEL
LIN {X 0,Y 456.725,Z 532.099,A -85,B 0,C 180,E1 -8218.365,E2 -8218.365} C_VEL
LIN {X 0,Y 457.051,Z 518.928,A -85,B 0,C 180,E1 -8218.774,E2 -8218.774} C_VEL
LIN {X 0,Y 457.425,Z 488.363,A -85,B 0,C 180,E1 -8219.293,E2 -8219.293} C_VEL
LIN {X 0,Y 457.961,Z 427.384,A -85,B 0,C 180,E1 -8220.269,E2 -8220.269} C_VEL
LIN {X 0,Y 454.752,Z 410.768,A -85,B 0,C 180,E1 -8220.702,E2 -8220.702} C_VEL
LIN {X 0,Y 454.698,Z 409.833,A -85,B 0,C 180,E1 -8220.796,E2 -8220.796} C_VEL
LIN {X 0,Y 455.505,Z 394.598,A -85,B 0,C 180,E1 -8224.007,E2 -8224.007} C_VEL
LIN {X 0,Y 454.995,Z 389.96,A -85,B 0,C 180,E1 -8225.049,E2 -8225.049} C_VEL
LIN {X 0,Y 453.476,Z 382.546,A -85,B 0,C 180,E1 -8226.843,E2 -8226.843} C_VEL
LIN {X 0,Y 453.53,Z 382.492,A -85,B 0,C 180,E1 -8229.444,E2 -8229.444} C_VEL
LIN {X 0,Y 453.487,Z 382.496,A -85,B 0,C 180,E1 -8232.991,E2 -8232.991} C_VEL
LIN {X 0,Y 453.472,Z 382.497,A -85,B 0,C 180,E1 -8235.78,E2 -8235.78} C_VEL
LIN {X 0,Y 453.491,Z 382.489,A -85,B 0,C 180,E1 -8238.211,E2 -8238.211} C_VEL
LIN {X 0,Y 453.527,Z 382.49,A -85,B 0,C 180,E1 -8240.787,E2 -8240.787} C_VEL
LIN {X 0,Y 453.451,Z 382.497,A -85,B 0,C 180,E1 -8243.917,E2 -8243.917} C_VEL
LIN {X 0,Y 453.476,Z 382.501,A -85,B 0,C 180,E1 -8247.151,E2 -8247.151} C_VEL
LIN {X 0,Y 453.506,Z 382.482,A -85,B 0,C 180,E1 -8250.271,E2 -8250.271} C_VEL
LIN {X 0,Y 453.506,Z 382.495,A -85,B 0,C 180,E1 -8253.294,E2 -8253.294} C_VEL
LIN {X 0,Y 453.496,Z 382.493,A -85,B 0,C 180,E1 -8256.238,E2 -8256.238} C_VEL
LIN {X 0,Y 453.499,Z 382.498,A -85,B 0,C 180,E1 -8259.118,E2 -8259.118} C_VEL
LIN {X 0,Y 453.503,Z 382.488,A -85,B 0,C 180,E1 -8261.944,E2 -8261.944} C_VEL
LIN {X 0,Y 453.531,Z 382.493,A -85,B 0,C 180,E1 -8264.726,E2 -8264.726} C_VEL
LIN {X 0,Y 453.593,Z 382.482,A -85,B 0,C 180,E1 -8267.472,E2 -8267.472} C_VEL
LIN {X 0,Y 453.585,Z 382.486,A -85,B 0,C 180,E1 -8271.087,E2 -8271.087} C_VEL
LIN {X 0,Y 453.671,Z 382.466,A -85,B 0,C 180,E1 -8273.775,E2 -8273.775} C_VEL
LIN {X 0,Y 453.765,Z 382.459,A -85,B 0,C 180,E1 -8277.337,E2 -8277.337} C_VEL
LIN {X 0,Y 453.815,Z 382.449,A -85,B 0,C 180,E1 -8280,E2 -8280} C_VEL
LIN {X 0,Y 453.758,Z 382.464,A -85,B 0,C 180,E1 -8282.663,E2 -8282.663} C_VEL
LIN {X 0,Y 453.671,Z 382.471,A -85,B 0,C 180,E1 -8286.225,E2 -8286.225} C_VEL
LIN {X 0,Y 453.585,Z 382.481,A -85,B 0,C 180,E1 -8288.914,E2 -8288.914} C_VEL
LIN {X 0,Y 453.593,Z 382.485,A -85,B 0,C 180,E1 -8292.551,E2 -8292.551} C_VEL
LIN {X 0,Y 453.536,Z 382.489,A -85,B 0,C 180,E1 -8296.196,E2 -8296.196} C_VEL
LIN {X 0,Y 453.512,Z 382.493,A -85,B 0,C 180,E1 -8299.041,E2 -8299.041} C_VEL
LIN {X 0,Y 453.471,Z 382.493,A -85,B 0,C 180,E1 -8301.837,E2 -8301.837} C_VEL
LIN {X 0,Y 453.508,Z 382.497,A -85,B 0,C 180,E1 -8304.735,E2 -8304.735} C_VEL
LIN {X 0,Y 453.53,Z 382.487,A -85,B 0,C 180,E1 -8307.962,E2 -8307.962} C_VEL
LIN {X 0,Y 453.46,Z 382.496,A -85,B 0,C 180,E1 -8311.526,E2 -8311.526} C_VEL
LIN {X 0,Y 453.483,Z 382.499,A -85,B 0,C 180,E1 -8314.779,E2 -8314.779} C_VEL
LIN {X 0,Y 453.478,Z 382.497,A -85,B 0,C 180,E1 -8318.31,E2 -8318.31} C_VEL
LIN {X 0,Y 453.511,Z 382.487,A -85,B 0,C 180,E1 -8320.607,E2 -8320.607} C_VEL
LIN {X 0,Y 453.478,Z 382.495,A -85,B 0,C 180,E1 -8323.249,E2 -8323.249} C_VEL
LIN {X 0,Y 453.469,Z 382.493,A -85,B 0,C 180,E1 -8325.781,E2 -8325.781} C_VEL
LIN {X 0,Y 453.478,Z 382.498,A -85,B 0,C 180,E1 -8328.21,E2 -8328.21} C_VEL
LIN {X 0,Y 453.507,Z 382.493,A -85,B 0,C 180,E1 -8330.792,E2 -8330.792} C_VEL
LIN {X 0,Y 453.455,Z 382.495,A -85,B 0,C 180,E1 -8333.918,E2 -8333.918} C_VEL
LIN {X 0,Y 453.482,Z 382.497,A -85,B 0,C 180,E1 -8337.152,E2 -8337.152} C_VEL
LIN {X 0,Y 453.475,Z 382.498,A -85,B 0,C 180,E1 -8340.269,E2 -8340.269} C_VEL
LIN {X 0,Y 453.514,Z 382.494,A -85,B 0,C 180,E1 -8343.295,E2 -8343.295} C_VEL
LIN {X 0,Y 453.553,Z 382.591,A -85,B 0,C 180,E1 -8344.349,E2 -8344.349} C_VEL
LIN {X 0,Y 455.56,Z 392.685,A -85,B 0,C 180,E1 -8346.594,E2 -8346.594} C_VEL
LIN {X 0,Y 455.976,Z 396.233,A -85,B 0,C 180,E1 -8347.337,E2 -8347.337} C_VEL
LIN {X 0,Y 454.889,Z 415.273,A -85,B 0,C 180,E1 -8351.069,E2 -8351.069} C_VEL
LIN {X 0,Y 454.577,Z 421.837,A -85,B 0,C 180,E1 -8352.303,E2 -8352.303} C_VEL
LIN {X 0,Y 455.632,Z 427.63,A -85,B 0,C 180,E1 -8352.481,E2 -8352.481} C_VEL
LIN {X 0,Y 457.924,Z 441.993,A -85,B 0,C 180,E1 -8352.816,E2 -8352.816} C_VEL
LIN {X 0,Y 457.049,Z 530.201,A -85,B 0,C 180,E1 -8354.247,E2 -8354.247} C_VEL
LIN {X 0,Y 456.645,Z 543.986,A -85,B 0,C 180,E1 -8354.662,E2 -8354.662} C_VEL
LIN {X 0,Y 456.157,Z 556.361,A -85,B 0,C 180,E1 -8355.216,E2 -8355.216} C_VEL
LIN {X 0,Y 455.57,Z 568.21,A -85,B 0,C 180,E1 -8355.938,E2 -8355.938} C_VEL
LIN {X 0,Y 454.919,Z 580.418,A -85,B 0,C 180,E1 -8356.901,E2 -8356.901} C_VEL
LIN {X 0,Y 454.396,Z 590.87,A -85,B 0,C 180,E1 -8357.948,E2 -8357.948} C_VEL
LIN {X 0,Y 453.815,Z 599.925,A -85,B 0,C 180,E1 -8359.065,E2 -8359.065} C_VEL
LIN {X 0,Y 453.341,Z 608.77,A -85,B 0,C 180,E1 -8360.407,E2 -8360.407} C_VEL
LIN {X 0,Y 452.968,Z 615.877,A -85,B 0,C 180,E1 -8361.749,E2 -8361.749} C_VEL
LIN {X 0,Y 452.76,Z 620.687,A -85,B 0,C 180,E1 -8362.867,E2 -8362.867} C_VEL
LIN {X 0,Y 452.613,Z 625.356,A -85,B 0,C 180,E1 -8364.208,E2 -8364.208} C_VEL
LIN {X 0,Y 452.489,Z 628.921,A -85,B 0,C 180,E1 -8365.546,E2 -8365.546} C_VEL
LIN {X 0,Y 452.456,Z 630.754,A -85,B 0,C 180,E1 -8366.438,E2 -8366.438} C_VEL
LIN {X 0,Y 452.49,Z 632.13,A -85,B 0,C 180,E1 -8367.33,E2 -8367.33} C_VEL
LIN {X 0,Y 452.403,Z 633.706,A -85,B 0,C 180,E1 -8369.11,E2 -8369.11} C_VEL
LIN {X 0,Y 452.407,Z 633.903,A -85,B 0,C 180,E1 -8370,E2 -8370} C_VEL
LIN {X 0,Y 452.432,Z 633.053,A -85,B 0,C 180,E1 -8371.781,E2 -8371.781} C_VEL
LIN {X 0,Y 452.491,Z 632.049,A -85,B 0,C 180,E1 -8372.671,E2 -8372.671} C_VEL
LIN {X 0,Y 452.456,Z 630.632,A -85,B 0,C 180,E1 -8373.562,E2 -8373.562} C_VEL
LIN {X 0,Y 452.557,Z 627.678,A -85,B 0,C 180,E1 -8374.9,E2 -8374.9} C_VEL
LIN {X 0,Y 452.629,Z 623.048,A -85,B 0,C 180,E1 -8376.416,E2 -8376.416} C_VEL
LIN {X 0,Y 452.87,Z 617.507,A -85,B 0,C 180,E1 -8377.804,E2 -8377.804} C_VEL
LIN {X 0,Y 453.169,Z 610.775,A -85,B 0,C 180,E1 -8379.147,E2 -8379.147} C_VEL
LIN {X 0,Y 453.574,Z 602.415,A -85,B 0,C 180,E1 -8380.49,E2 -8380.49} C_VEL
LIN {X 0,Y 454.082,Z 593.8,A -85,B 0,C 180,E1 -8381.607,E2 -8381.607} C_VEL
LIN {X 0,Y 454.63,Z 583.816,A -85,B 0,C 180,E1 -8382.664,E2 -8382.664} C_VEL
LIN {X 0,Y 455.196,Z 572.619,A -85,B 0,C 180,E1 -8383.618,E2 -8383.618} C_VEL
LIN {X 0,Y 455.683,Z 560.918,A -85,B 0,C 180,E1 -8384.4,E2 -8384.4} C_VEL
LIN {X 0,Y 456.209,Z 548.742,A -85,B 0,C 180,E1 -8385.011,E2 -8385.011} C_VEL
LIN {X 0,Y 456.659,Z 535.461,A -85,B 0,C 180,E1 -8385.481,E2 -8385.481} C_VEL
LIN {X 0,Y 456.846,Z 522.385,A -85,B 0,C 180,E1 -8385.761,E2 -8385.761} C_VEL
LIN {X 0,Y 457.445,Z 440.72,A -85,B 0,C 180,E1 -8387.048,E2 -8387.048} C_VEL
LIN {X 0,Y 454.413,Z 422.129,A -85,B 0,C 180,E1 -8387.472,E2 -8387.472} C_VEL
LIN {X 0,Y 455.008,Z 408.091,A -85,B 0,C 180,E1 -8390.1,E2 -8390.1} C_VEL
LIN {X 0,Y 455.669,Z 394.693,A -85,B 0,C 180,E1 -8392.68,E2 -8392.68} C_VEL
LIN {X 0,Y 453.995,Z 384.848,A -85,B 0,C 180,E1 -8394.706,E2 -8394.706} C_VEL
LIN {X 0,Y 453.553,Z 382.526,A -85,B 0,C 180,E1 -8395.252,E2 -8395.252} C_VEL
LIN {X 0,Y 453.512,Z 382.493,A -85,B 0,C 180,E1 -8398.711,E2 -8398.711} C_VEL
LIN {X 0,Y 453.466,Z 382.499,A -85,B 0,C 180,E1 -8401.799,E2 -8401.799} C_VEL
LIN {X 0,Y 453.482,Z 382.496,A -85,B 0,C 180,E1 -8404.989,E2 -8404.989} C_VEL
LIN {X 0,Y 453.473,Z 382.495,A -85,B 0,C 180,E1 -8408.31,E2 -8408.31} C_VEL
LIN {X 0,Y 453.493,Z 382.493,A -85,B 0,C 180,E1 -8410.608,E2 -8410.608} C_VEL
LIN {X 0,Y 453.462,Z 382.502,A -85,B 0,C 180,E1 -8413.245,E2 -8413.245} C_VEL
LIN {X 0,Y 453.475,Z 382.497,A -85,B 0,C 180,E1 -8415.78,E2 -8415.78} C_VEL
LIN {X 0,Y 453.495,Z 382.494,A -85,B 0,C 180,E1 -8418.211,E2 -8418.211} C_VEL
LIN {X 0,Y 453.53,Z 382.49,A -85,B 0,C 180,E1 -8420.787,E2 -8420.787} C_VEL
LIN {X 0,Y 453.454,Z 382.499,A -85,B 0,C 180,E1 -8423.917,E2 -8423.917} C_VEL
LIN {X 0,Y 453.479,Z 382.5,A -85,B 0,C 180,E1 -8427.151,E2 -8427.151} C_VEL
LIN {X 0,Y 453.471,Z 382.497,A -85,B 0,C 180,E1 -8430.268,E2 -8430.268} C_VEL
LIN {X 0,Y 453.509,Z 382.495,A -85,B 0,C 180,E1 -8433.294,E2 -8433.294} C_VEL
LIN {X 0,Y 453.498,Z 382.494,A -85,B 0,C 180,E1 -8436.238,E2 -8436.238} C_VEL
LIN {X 0,Y 453.478,Z 382.5,A -85,B 0,C 180,E1 -8439.117,E2 -8439.117} C_VEL
LIN {X 0,Y 453.507,Z 382.494,A -85,B 0,C 180,E1 -8441.944,E2 -8441.944} C_VEL
LIN {X 0,Y 453.534,Z 382.491,A -85,B 0,C 180,E1 -8444.726,E2 -8444.726} C_VEL
LIN {X 0,Y 453.553,Z 382.488,A -85,B 0,C 180,E1 -8448.379,E2 -8448.379} C_VEL
LIN {X 0,Y 453.646,Z 382.477,A -85,B 0,C 180,E1 -8451.985,E2 -8451.985} C_VEL
LIN {X 0,Y 453.665,Z 382.475,A -85,B 0,C 180,E1 -8454.667,E2 -8454.667} C_VEL
LIN {X 0,Y 453.759,Z 382.462,A -85,B 0,C 180,E1 -8457.337,E2 -8457.337} C_VEL
LIN {X 0,Y 453.817,Z 382.456,A -85,B 0,C 180,E1 -8460,E2 -8460} C_VEL
LIN {X 0,Y 453.76,Z 382.464,A -85,B 0,C 180,E1 -8462.663,E2 -8462.663} C_VEL
LIN {X 0,Y 453.671,Z 382.473,A -85,B 0,C 180,E1 -8466.225,E2 -8466.225} C_VEL
LIN {X 0,Y 453.586,Z 382.485,A -85,B 0,C 180,E1 -8468.913,E2 -8468.913} C_VEL
LIN {X 0,Y 453.557,Z 382.488,A -85,B 0,C 180,E1 -8472.529,E2 -8472.529} C_VEL
LIN {X 0,Y 453.539,Z 382.49,A -85,B 0,C 180,E1 -8476.196,E2 -8476.196} C_VEL
LIN {X 0,Y 453.515,Z 382.493,A -85,B 0,C 180,E1 -8479.041,E2 -8479.041} C_VEL
LIN {X 0,Y 453.471,Z 382.499,A -85,B 0,C 180,E1 -8481.836,E2 -8481.836} C_VEL
LIN {X 0,Y 453.509,Z 382.494,A -85,B 0,C 180,E1 -8484.735,E2 -8484.735} C_VEL
LIN {X 0,Y 453.534,Z 382.49,A -85,B 0,C 180,E1 -8487.962,E2 -8487.962} C_VEL
LIN {X 0,Y 453.479,Z 382.497,A -85,B 0,C 180,E1 -8490.759,E2 -8490.759} C_VEL
LIN {X 0,Y 453.474,Z 382.498,A -85,B 0,C 180,E1 -8493.913,E2 -8493.913} C_VEL
LIN {X 0,Y 453.467,Z 382.5,A -85,B 0,C 180,E1 -8497.188,E2 -8497.188} C_VEL
LIN {X 0,Y 453.502,Z 382.497,A -85,B 0,C 180,E1 -8499.449,E2 -8499.449} C_VEL
LIN {X 0,Y 453.465,Z 382.499,A -85,B 0,C 180,E1 -8502.995,E2 -8502.995} C_VEL
LIN {X 0,Y 453.463,Z 382.499,A -85,B 0,C 180,E1 -8505.78,E2 -8505.78} C_VEL
LIN {X 0,Y 453.514,Z 382.495,A -85,B 0,C 180,E1 -8509.406,E2 -8509.406} C_VEL
LIN {X 0,Y 453.475,Z 382.497,A -85,B 0,C 180,E1 -8512.223,E2 -8512.223} C_VEL
LIN {X 0,Y 453.488,Z 382.5,A -85,B 0,C 180,E1 -8515.223,E2 -8515.223} C_VEL
LIN {X 0,Y 453.465,Z 382.497,A -85,B 0,C 180,E1 -8518.475,E2 -8518.475} C_VEL
LIN {X 0,Y 453.532,Z 382.488,A -85,B 0,C 180,E1 -8522.041,E2 -8522.041} C_VEL
LIN {X 0,Y 453.514,Z 382.495,A -85,B 0,C 180,E1 -8525.266,E2 -8525.266} C_VEL
LIN {X 0,Y 453.481,Z 382.495,A -85,B 0,C 180,E1 -8528.415,E2 -8528.415} C_VEL
LIN {X 0,Y 453.523,Z 382.496,A -85,B 0,C 180,E1 -8531.009,E2 -8531.009} C_VEL
LIN {X 0,Y 453.57,Z 382.483,A -85,B 0,C 180,E1 -8533.88,E2 -8533.88} C_VEL
LIN {X 0,Y 453.565,Z 382.488,A -85,B 0,C 180,E1 -8537.471,E2 -8537.471} C_VEL
LIN {X 0,Y 453.588,Z 382.684,A -85,B 0,C 180,E1 -8539.736,E2 -8539.736} C_VEL
LIN {X 0,Y 455.116,Z 390.945,A -85,B 0,C 180,E1 -8541.597,E2 -8541.597} C_VEL
LIN {X 0,Y 454.983,Z 396.157,A -85,B 0,C 180,E1 -8542.696,E2 -8542.696} C_VEL
LIN {X 0,Y 454.119,Z 398.291,A -85,B 0,C 180,E1 -8543.109,E2 -8543.109} C_VEL
LIN {X 0,Y 448.088,Z 405.387,A -85,B 0,C 180,E1 -8544.357,E2 -8544.357} C_VEL
LIN {X 0,Y 447.516,Z 407.488,A -85,B 0,C 180,E1 -8544.78,E2 -8544.78} C_VEL
LIN {X 0,Y 447.538,Z 410.378,A -85,B 0,C 180,E1 -8545.327,E2 -8545.327} C_VEL
LIN {X 0,Y 448.518,Z 416.301,A -85,B 0,C 180,E1 -8545.496,E2 -8545.496} C_VEL
LIN {X 0,Y 450.664,Z 427.513,A -85,B 0,C 180,E1 -8545.752,E2 -8545.752} C_VEL
LIN {X 0,Y 449.915,Z 517.149,A -85,B 0,C 180,E1 -8547.202,E2 -8547.202} C_VEL
LIN {X 0,Y 449.553,Z 530.386,A -85,B 0,C 180,E1 -8547.592,E2 -8547.592} C_VEL
LIN {X 0,Y 449.126,Z 543.048,A -85,B 0,C 180,E1 -8548.15,E2 -8548.15} C_VEL
LIN {X 0,Y 448.605,Z 555.127,A -85,B 0,C 180,E1 -8548.878,E2 -8548.878} C_VEL
LIN {X 0,Y 447.962,Z 566.61,A -85,B 0,C 180,E1 -8549.775,E2 -8549.775} C_VEL
LIN {X 0,Y 447.342,Z 576.959,A -85,B 0,C 180,E1 -8550.787,E2 -8550.787} C_VEL
LIN {X 0,Y 446.894,Z 585.416,A -85,B 0,C 180,E1 -8551.802,E2 -8551.802} C_VEL
LIN {X 0,Y 446.434,Z 593.24,A -85,B 0,C 180,E1 -8552.932,E2 -8552.932} C_VEL
LIN {X 0,Y 446.053,Z 600.887,A -85,B 0,C 180,E1 -8554.292,E2 -8554.292} C_VEL
LIN {X 0,Y 445.776,Z 606.139,A -85,B 0,C 180,E1 -8555.428,E2 -8555.428} C_VEL
LIN {X 0,Y 445.631,Z 611.22,A -85,B 0,C 180,E1 -8556.792,E2 -8556.792} C_VEL
LIN {X 0,Y 445.475,Z 615.182,A -85,B 0,C 180,E1 -8558.162,E2 -8558.162} C_VEL
LIN {X 0,Y 445.355,Z 617.224,A -85,B 0,C 180,E1 -8559.079,E2 -8559.079} C_VEL
LIN {X 0,Y 445.3,Z 618.845,A -85,B 0,C 180,E1 -8559.997,E2 -8559.997} C_VEL
LIN {X 0,Y 445.304,Z 620.053,A -85,B 0,C 180,E1 -8560.917,E2 -8560.917} C_VEL
LIN {X 0,Y 445.337,Z 620.849,A -85,B 0,C 180,E1 -8561.919,E2 -8561.919} C_VEL
LIN {X 0,Y 445.252,Z 621.121,A -85,B 0,C 180,E1 -8563.695,E2 -8563.695} C_VEL
LIN {X 0,Y 445.268,Z 620.658,A -85,B 0,C 180,E1 -8564.627,E2 -8564.627} C_VEL
LIN {X 0,Y 445.301,Z 619.581,A -85,B 0,C 180,E1 -8565.69,E2 -8565.69} C_VEL
LIN {X 0,Y 445.39,Z 616.632,A -85,B 0,C 180,E1 -8567.446,E2 -8567.446} C_VEL
LIN {X 0,Y 445.56,Z 613.095,A -85,B 0,C 180,E1 -8568.843,E2 -8568.843} C_VEL
LIN {X 0,Y 445.783,Z 608.207,A -85,B 0,C 180,E1 -8570.294,E2 -8570.294} C_VEL
LIN {X 0,Y 446.156,Z 601.314,A -85,B 0,C 180,E1 -8571.869,E2 -8571.869} C_VEL
LIN {X 0,Y 446.579,Z 594.18,A -85,B 0,C 180,E1 -8573.168,E2 -8573.168} C_VEL
LIN {X 0,Y 447.071,Z 586.278,A -85,B 0,C 180,E1 -8574.346,E2 -8574.346} C_VEL
LIN {X 0,Y 447.606,Z 577.207,A -85,B 0,C 180,E1 -8575.456,E2 -8575.456} C_VEL
LIN {X 0,Y 448.187,Z 567.705,A -85,B 0,C 180,E1 -8576.405,E2 -8576.405} C_VEL
LIN {X 0,Y 448.882,Z 555.484,A -85,B 0,C 180,E1 -8577.381,E2 -8577.381} C_VEL
LIN {X 0,Y 449.496,Z 543.789,A -85,B 0,C 180,E1 -8578.099,E2 -8578.099} C_VEL
LIN {X 0,Y 449.954,Z 531.123,A -85,B 0,C 180,E1 -8578.672,E2 -8578.672} C_VEL
LIN {X 0,Y 450.322,Z 518.232,A -85,B 0,C 180,E1 -8579.065,E2 -8579.065} C_VEL
LIN {X 0,Y 451.224,Z 428.258,A -85,B 0,C 180,E1 -8580.549,E2 -8580.549} C_VEL
LIN {X 0,Y 447.98,Z 411.54,A -85,B 0,C 180,E1 -8580.985,E2 -8580.985} C_VEL
LIN {X 0,Y 447.794,Z 410.125,A -85,B 0,C 180,E1 -8581.078,E2 -8581.078} C_VEL
LIN {X 0,Y 448.562,Z 396.266,A -85,B 0,C 180,E1 -8584.037,E2 -8584.037} C_VEL
LIN {X 0,Y 448.273,Z 392.427,A -85,B 0,C 180,E1 -8584.906,E2 -8584.906} C_VEL
LIN {X 0,Y 446.458,Z 383.423,A -85,B 0,C 180,E1 -8587.109,E2 -8587.109} C_VEL
LIN {X 0,Y 446.465,Z 383.372,A -85,B 0,C 180,E1 -8590.194,E2 -8590.194} C_VEL
LIN {X 0,Y 446.442,Z 383.376,A -85,B 0,C 180,E1 -8593.602,E2 -8593.602} C_VEL
LIN {X 0,Y 446.442,Z 383.373,A -85,B 0,C 180,E1 -8596.396,E2 -8596.396} C_VEL
LIN {X 0,Y 446.463,Z 383.37,A -85,B 0,C 180,E1 -8599.804,E2 -8599.804} C_VEL
LIN {X 0,Y 446.429,Z 383.371,A -85,B 0,C 180,E1 -8602.123,E2 -8602.123} C_VEL
LIN {X 0,Y 446.424,Z 383.37,A -85,B 0,C 180,E1 -8605.476,E2 -8605.476} C_VEL
LIN {X 0,Y 446.427,Z 383.377,A -85,B 0,C 180,E1 -8608.7,E2 -8608.7} C_VEL
LIN {X 0,Y 446.477,Z 383.366,A -85,B 0,C 180,E1 -8611.821,E2 -8611.821} C_VEL
LIN {X 0,Y 446.451,Z 383.373,A -85,B 0,C 180,E1 -8614.847,E2 -8614.847} C_VEL
LIN {X 0,Y 446.461,Z 383.365,A -85,B 0,C 180,E1 -8618.238,E2 -8618.238} C_VEL
LIN {X 0,Y 446.449,Z 383.367,A -85,B 0,C 180,E1 -8621.649,E2 -8621.649} C_VEL
LIN {X 0,Y 446.499,Z 383.366,A -85,B 0,C 180,E1 -8624.479,E2 -8624.479} C_VEL
LIN {X 0,Y 446.531,Z 383.36,A -85,B 0,C 180,E1 -8628.193,E2 -8628.193} C_VEL
LIN {X 0,Y 446.591,Z 383.352,A -85,B 0,C 180,E1 -8631.858,E2 -8631.858} C_VEL
LIN {X 0,Y 446.64,Z 383.345,A -85,B 0,C 180,E1 -8634.583,E2 -8634.583} C_VEL
LIN {X 0,Y 446.709,Z 383.338,A -85,B 0,C 180,E1 -8637.295,E2 -8637.295} C_VEL
LIN {X 0,Y 446.785,Z 383.325,A -85,B 0,C 180,E1 -8640,E2 -8640} C_VEL
LIN {X 0,Y 446.702,Z 383.342,A -85,B 0,C 180,E1 -8642.705,E2 -8642.705} C_VEL
LIN {X 0,Y 446.64,Z 383.348,A -85,B 0,C 180,E1 -8646.324,E2 -8646.324} C_VEL
LIN {X 0,Y 446.531,Z 383.36,A -85,B 0,C 180,E1 -8649.056,E2 -8649.056} C_VEL
LIN {X 0,Y 446.525,Z 383.362,A -85,B 0,C 180,E1 -8652.73,E2 -8652.73} C_VEL
LIN {X 0,Y 446.481,Z 383.37,A -85,B 0,C 180,E1 -8656.46,E2 -8656.46} C_VEL
LIN {X 0,Y 446.461,Z 383.368,A -85,B 0,C 180,E1 -8659.304,E2 -8659.304} C_VEL
LIN {X 0,Y 446.413,Z 383.375,A -85,B 0,C 180,E1 -8662.2,E2 -8662.2} C_VEL
LIN {X 0,Y 446.451,Z 383.371,A -85,B 0,C 180,E1 -8665.153,E2 -8665.153} C_VEL
LIN {X 0,Y 446.477,Z 383.367,A -85,B 0,C 180,E1 -8668.179,E2 -8668.179} C_VEL
LIN {X 0,Y 446.413,Z 383.374,A -85,B 0,C 180,E1 -8671.776,E2 -8671.776} C_VEL
LIN {X 0,Y 446.424,Z 383.376,A -85,B 0,C 180,E1 -8674.524,E2 -8674.524} C_VEL
LIN {X 0,Y 446.431,Z 383.372,A -85,B 0,C 180,E1 -8678.084,E2 -8678.084} C_VEL
LIN {X 0,Y 446.442,Z 383.362,A -85,B 0,C 180,E1 -8680.921,E2 -8680.921} C_VEL
LIN {X 0,Y 446.441,Z 383.372,A -85,B 0,C 180,E1 -8683.841,E2 -8683.841} C_VEL
LIN {X 0,Y 446.417,Z 383.371,A -85,B 0,C 180,E1 -8686.401,E2 -8686.401} C_VEL
LIN {X 0,Y 446.445,Z 383.369,A -85,B 0,C 180,E1 -8689.804,E2 -8689.804} C_VEL
LIN {X 0,Y 446.425,Z 383.378,A -85,B 0,C 180,E1 -8692.124,E2 -8692.124} C_VEL
LIN {X 0,Y 446.429,Z 383.373,A -85,B 0,C 180,E1 -8695.478,E2 -8695.478} C_VEL
LIN {X 0,Y 446.416,Z 383.378,A -85,B 0,C 180,E1 -8698.701,E2 -8698.701} C_VEL
LIN {X 0,Y 446.484,Z 383.369,A -85,B 0,C 180,E1 -8701.822,E2 -8701.822} C_VEL
LIN {X 0,Y 446.507,Z 383.533,A -85,B 0,C 180,E1 -8704.102,E2 -8704.102} C_VEL
LIN {X 0,Y 448.821,Z 395.161,A -85,B 0,C 180,E1 -8706.711,E2 -8706.711} C_VEL
LIN {X 0,Y 448.947,Z 399.45,A -85,B 0,C 180,E1 -8707.599,E2 -8707.599} C_VEL
LIN {X 0,Y 447.852,Z 417.739,A -85,B 0,C 180,E1 -8711.235,E2 -8711.235} C_VEL
LIN {X 0,Y 447.666,Z 421.808,A -85,B 0,C 180,E1 -8711.994,E2 -8711.994} C_VEL
LIN {X 0,Y 449.122,Z 429.71,A -85,B 0,C 180,E1 -8712.229,E2 -8712.229} C_VEL
LIN {X 0,Y 451.208,Z 442.748,A -85,B 0,C 180,E1 -8712.539,E2 -8712.539} C_VEL
LIN {X 0,Y 450.283,Z 530.094,A -85,B 0,C 180,E1 -8713.975,E2 -8713.975} C_VEL
LIN {X 0,Y 449.86,Z 543.867,A -85,B 0,C 180,E1 -8714.396,E2 -8714.396} C_VEL
LIN {X 0,Y 449.384,Z 555.689,A -85,B 0,C 180,E1 -8714.93,E2 -8714.93} C_VEL
LIN {X 0,Y 448.796,Z 566.896,A -85,B 0,C 180,E1 -8715.606,E2 -8715.606} C_VEL
LIN {X 0,Y 448.13,Z 578.32,A -85,B 0,C 180,E1 -8716.494,E2 -8716.494} C_VEL
LIN {X 0,Y 447.539,Z 588.936,A -85,B 0,C 180,E1 -8717.531,E2 -8717.531} C_VEL
LIN {X 0,Y 446.931,Z 598.36,A -85,B 0,C 180,E1 -8718.664,E2 -8718.664} C_VEL
LIN {X 0,Y 446.4,Z 607.45,A -85,B 0,C 180,E1 -8720.028,E2 -8720.028} C_VEL
LIN {X 0,Y 445.985,Z 614.782,A -85,B 0,C 180,E1 -8721.391,E2 -8721.391} C_VEL
LIN {X 0,Y 445.69,Z 620.671,A -85,B 0,C 180,E1 -8722.753,E2 -8722.753} C_VEL
LIN {X 0,Y 445.514,Z 624.668,A -85,B 0,C 180,E1 -8723.907,E2 -8723.907} C_VEL
LIN {X 0,Y 445.416,Z 628.868,A -85,B 0,C 180,E1 -8725.475,E2 -8725.475} C_VEL
LIN {X 0,Y 445.356,Z 630.686,A -85,B 0,C 180,E1 -8726.381,E2 -8726.381} C_VEL
LIN {X 0,Y 445.398,Z 632.054,A -85,B 0,C 180,E1 -8727.287,E2 -8727.287} C_VEL
LIN {X 0,Y 445.315,Z 633.616,A -85,B 0,C 180,E1 -8729.096,E2 -8729.096} C_VEL
LIN {X 0,Y 445.316,Z 633.8,A -85,B 0,C 180,E1 -8730,E2 -8730} C_VEL
LIN {X 0,Y 445.352,Z 632.936,A -85,B 0,C 180,E1 -8731.809,E2 -8731.809} C_VEL
LIN {X 0,Y 445.398,Z 631.924,A -85,B 0,C 180,E1 -8732.713,E2 -8732.713} C_VEL
LIN {X 0,Y 445.356,Z 630.493,A -85,B 0,C 180,E1 -8733.619,E2 -8733.619} C_VEL
LIN {X 0,Y 445.489,Z 627.526,A -85,B 0,C 180,E1 -8734.978,E2 -8734.978} C_VEL
LIN {X 0,Y 445.611,Z 622.053,A -85,B 0,C 180,E1 -8736.748,E2 -8736.748} C_VEL
LIN {X 0,Y 445.856,Z 616.298,A -85,B 0,C 180,E1 -8738.156,E2 -8738.156} C_VEL
LIN {X 0,Y 446.222,Z 609.306,A -85,B 0,C 180,E1 -8739.519,E2 -8739.519} C_VEL
LIN {X 0,Y 446.663,Z 600.528,A -85,B 0,C 180,E1 -8740.884,E2 -8740.884} C_VEL
LIN {X 0,Y 447.277,Z 590.555,A -85,B 0,C 180,E1 -8742.132,E2 -8742.132} C_VEL
LIN {X 0,Y 447.835,Z 579.847,A -85,B 0,C 180,E1 -8743.201,E2 -8743.201} C_VEL
LIN {X 0,Y 448.405,Z 569.095,A -85,B 0,C 180,E1 -8744.06,E2 -8744.06} C_VEL
LIN {X 0,Y 448.929,Z 557.383,A -85,B 0,C 180,E1 -8744.796,E2 -8744.796} C_VEL
LIN {X 0,Y 449.465,Z 544.659,A -85,B 0,C 180,E1 -8745.386,E2 -8745.386} C_VEL
LIN {X 0,Y 449.84,Z 532.228,A -85,B 0,C 180,E1 -8745.78,E2 -8745.78} C_VEL
LIN {X 0,Y 450.086,Z 511.735,A -85,B 0,C 180,E1 -8746.149,E2 -8746.149} C_VEL
LIN {X 0,Y 450.537,Z 441.063,A -85,B 0,C 180,E1 -8747.282,E2 -8747.282} C_VEL
LIN {X 0,Y 447.429,Z 421.951,A -85,B 0,C 180,E1 -8747.73,E2 -8747.73} C_VEL
LIN {X 0,Y 448.092,Z 407.832,A -85,B 0,C 180,E1 -8750.424,E2 -8750.424} C_VEL
LIN {X 0,Y 448.7,Z 396.253,A -85,B 0,C 180,E1 -8752.689,E2 -8752.689} C_VEL
LIN {X 0,Y 447.697,Z 389.486,A -85,B 0,C 180,E1 -8754.088,E2 -8754.088} C_VEL
LIN {X 0,Y 446.546,Z 383.425,A -85,B 0,C 180,E1 -8755.427,E2 -8755.427} C_VEL
LIN {X 0,Y 446.486,Z 383.369,A -85,B 0,C 180,E1 -8758.178,E2 -8758.178} C_VEL
LIN {X 0,Y 446.421,Z 383.377,A -85,B 0,C 180,E1 -8761.775,E2 -8761.775} C_VEL
LIN {X 0,Y 446.431,Z 383.372,A -85,B 0,C 180,E1 -8764.522,E2 -8764.522} C_VEL
LIN {X 0,Y 446.431,Z 383.373,A -85,B 0,C 180,E1 -8768.081,E2 -8768.081} C_VEL
LIN {X 0,Y 446.427,Z 383.375,A -85,B 0,C 180,E1 -8770.917,E2 -8770.917} C_VEL
LIN {X 0,Y 446.421,Z 383.376,A -85,B 0,C 180,E1 -8773.843,E2 -8773.843} C_VEL
LIN {X 0,Y 446.445,Z 383.372,A -85,B 0,C 180,E1 -8776.396,E2 -8776.396} C_VEL
LIN {X 0,Y 446.467,Z 383.37,A -85,B 0,C 180,E1 -8779.804,E2 -8779.804} C_VEL
LIN {X 0,Y 446.431,Z 383.374,A -85,B 0,C 180,E1 -8782.123,E2 -8782.123} C_VEL
LIN {X 0,Y 446.427,Z 383.377,A -85,B 0,C 180,E1 -8785.477,E2 -8785.477} C_VEL
LIN {X 0,Y 446.412,Z 383.377,A -85,B 0,C 180,E1 -8788.699,E2 -8788.699} C_VEL
LIN {X 0,Y 446.48,Z 383.368,A -85,B 0,C 180,E1 -8791.821,E2 -8791.821} C_VEL
LIN {X 0,Y 446.454,Z 383.373,A -85,B 0,C 180,E1 -8794.847,E2 -8794.847} C_VEL
LIN {X 0,Y 446.443,Z 383.373,A -85,B 0,C 180,E1 -8798.245,E2 -8798.245} C_VEL
LIN {X 0,Y 446.452,Z 383.372,A -85,B 0,C 180,E1 -8801.649,E2 -8801.649} C_VEL
LIN {X 0,Y 446.502,Z 383.366,A -85,B 0,C 180,E1 -8804.479,E2 -8804.479} C_VEL
LIN {X 0,Y 446.511,Z 383.365,A -85,B 0,C 180,E1 -8808.193,E2 -8808.193} C_VEL
LIN {X 0,Y 446.594,Z 383.356,A -85,B 0,C 180,E1 -8811.858,E2 -8811.858} C_VEL
LIN {X 0,Y 446.639,Z 383.349,A -85,B 0,C 180,E1 -8814.582,E2 -8814.582} C_VEL
LIN {X 0,Y 446.703,Z 383.342,A -85,B 0,C 180,E1 -8817.295,E2 -8817.295} C_VEL
LIN {X 0,Y 446.787,Z 383.331,A -85,B 0,C 180,E1 -8820,E2 -8820} C_VEL
LIN {X 0,Y 446.704,Z 383.343,A -85,B 0,C 180,E1 -8822.705,E2 -8822.705} C_VEL
LIN {X 0,Y 446.64,Z 383.349,A -85,B 0,C 180,E1 -8826.324,E2 -8826.324} C_VEL
LIN {X 0,Y 446.532,Z 383.363,A -85,B 0,C 180,E1 -8829.055,E2 -8829.055} C_VEL
LIN {X 0,Y 446.515,Z 383.366,A -85,B 0,C 180,E1 -8832.73,E2 -8832.73} C_VEL
LIN {X 0,Y 446.49,Z 383.368,A -85,B 0,C 180,E1 -8836.228,E2 -8836.228} C_VEL
LIN {X 0,Y 446.464,Z 383.372,A -85,B 0,C 180,E1 -8839.303,E2 -8839.303} C_VEL
LIN {X 0,Y 446.413,Z 383.377,A -85,B 0,C 180,E1 -8842.2,E2 -8842.2} C_VEL
LIN {X 0,Y 446.453,Z 383.373,A -85,B 0,C 180,E1 -8845.153,E2 -8845.153} C_VEL
LIN {X 0,Y 446.48,Z 383.369,A -85,B 0,C 180,E1 -8848.179,E2 -8848.179} C_VEL
LIN {X 0,Y 446.426,Z 383.377,A -85,B 0,C 180,E1 -8851.3,E2 -8851.3} C_VEL
LIN {X 0,Y 446.426,Z 383.376,A -85,B 0,C 180,E1 -8854.523,E2 -8854.523} C_VEL
LIN {X 0,Y 446.427,Z 383.375,A -85,B 0,C 180,E1 -8858.082,E2 -8858.082} C_VEL
LIN {X 0,Y 446.424,Z 383.376,A -85,B 0,C 180,E1 -8860.918,E2 -8860.918} C_VEL
LIN {X 0,Y 446.42,Z 383.376,A -85,B 0,C 180,E1 -8863.844,E2 -8863.844} C_VEL
LIN {X 0,Y 446.397,Z 383.379,A -85,B 0,C 180,E1 -8866.404,E2 -8866.404} C_VEL
LIN {X 0,Y 446.466,Z 383.37,A -85,B 0,C 180,E1 -8869.805,E2 -8869.805} C_VEL
LIN {X 0,Y 446.432,Z 383.374,A -85,B 0,C 180,E1 -8872.124,E2 -8872.124} C_VEL
LIN {X 0,Y 446.43,Z 383.376,A -85,B 0,C 180,E1 -8875.478,E2 -8875.478} C_VEL
LIN {X 0,Y 446.416,Z 383.376,A -85,B 0,C 180,E1 -8878.7,E2 -8878.7} C_VEL
LIN {X 0,Y 446.484,Z 383.366,A -85,B 0,C 180,E1 -8881.822,E2 -8881.822} C_VEL
LIN {X 0,Y 446.458,Z 383.373,A -85,B 0,C 180,E1 -8884.848,E2 -8884.848} C_VEL
LIN {X 0,Y 446.449,Z 383.37,A -85,B 0,C 180,E1 -8888.245,E2 -8888.245} C_VEL
LIN {X 0,Y 446.458,Z 383.37,A -85,B 0,C 180,E1 -8891.649,E2 -8891.649} C_VEL
LIN {X 0,Y 446.509,Z 383.364,A -85,B 0,C 180,E1 -8894.48,E2 -8894.48} C_VEL
LIN {X 0,Y 446.52,Z 383.366,A -85,B 0,C 180,E1 -8898.193,E2 -8898.193} C_VEL
LIN {X 0,Y 446.562,Z 383.596,A -85,B 0,C 180,E1 -8899.573,E2 -8899.573} C_VEL
LIN {X 0,Y 448.13,Z 392.028,A -85,B 0,C 180,E1 -8901.495,E2 -8901.495} C_VEL
LIN {X 0,Y 447.966,Z 400.191,A -85,B 0,C 180,E1 -8903.243,E2 -8903.243} C_VEL
LIN {X 0,Y 447.71,Z 403.4,A -85,B 0,C 180,E1 -8903.917,E2 -8903.917} C_VEL
LIN {X 0,Y 447.516,Z 407.488,A -85,B 0,C 180,E1 -8904.78,E2 -8904.78} C_VEL
LIN {X 0,Y 447.096,Z 409.343,A -85,B 0,C 180,E1 -8905.031,E2 -8905.031} C_VEL
LIN {X 0,Y 445.554,Z 412.484,A -85,B 0,C 180,E1 -8905.218,E2 -8905.218} C_VEL
LIN {X 0,Y 443.155,Z 416.995,A -85,B 0,C 180,E1 -8905.298,E2 -8905.298} C_VEL
LIN {X 0,Y 441.781,Z 421.47,A -85,B 0,C 180,E1 -8905.334,E2 -8905.334} C_VEL
LIN {X 0,Y 441.784,Z 425.264,A -85,B 0,C 180,E1 -8905.396,E2 -8905.396} C_VEL
LIN {X 0,Y 443.806,Z 437.109,A -85,B 0,C 180,E1 -8905.663,E2 -8905.663} C_VEL
LIN {X 0,Y 443.817,Z 438.209,A -85,B 0,C 180,E1 -8905.681,E2 -8905.681} C_VEL
LIN {X 0,Y 443.044,Z 517.516,A -85,B 0,C 180,E1 -8906.988,E2 -8906.988} C_VEL
LIN {X 0,Y 442.662,Z 530.667,A -85,B 0,C 180,E1 -8907.384,E2 -8907.384} C_VEL
LIN {X 0,Y 442.207,Z 543.287,A -85,B 0,C 180,E1 -8907.951,E2 -8907.951} C_VEL
LIN {X 0,Y 441.694,Z 554.539,A -85,B 0,C 180,E1 -8908.632,E2 -8908.632} C_VEL
LIN {X 0,Y 441.052,Z 566.152,A -85,B 0,C 180,E1 -8909.543,E2 -8909.543} C_VEL
LIN {X 0,Y 440.379,Z 576.609,A -85,B 0,C 180,E1 -8910.571,E2 -8910.571} C_VEL
LIN {X 0,Y 439.913,Z 585.145,A -85,B 0,C 180,E1 -8911.602,E2 -8911.602} C_VEL
LIN {X 0,Y 439.403,Z 593.041,A -85,B 0,C 180,E1 -8912.75,E2 -8912.75} C_VEL
LIN {X 0,Y 439.012,Z 600.763,A -85,B 0,C 180,E1 -8914.131,E2 -8914.131} C_VEL
LIN {X 0,Y 438.702,Z 606.964,A -85,B 0,C 180,E1 -8915.515,E2 -8915.515} C_VEL
LIN {X 0,Y 438.52,Z 611.897,A -85,B 0,C 180,E1 -8916.903,E2 -8916.903} C_VEL
LIN {X 0,Y 438.362,Z 615.716,A -85,B 0,C 180,E1 -8918.296,E2 -8918.296} C_VEL
LIN {X 0,Y 438.24,Z 617.689,A -85,B 0,C 180,E1 -8919.228,E2 -8919.228} C_VEL
LIN {X 0,Y 438.223,Z 619.237,A -85,B 0,C 180,E1 -8920.16,E2 -8920.16} C_VEL
LIN {X 0,Y 438.248,Z 620.977,A -85,B 0,C 180,E1 -8921.977,E2 -8921.977} C_VEL
LIN {X 0,Y 438.157,Z 621.297,A -85,B 0,C 180,E1 -8922.976,E2 -8922.976} C_VEL
LIN {X 0,Y 438.147,Z 621.172,A -85,B 0,C 180,E1 -8923.922,E2 -8923.922} C_VEL
LIN {X 0,Y 438.168,Z 620.592,A -85,B 0,C 180,E1 -8924.87,E2 -8924.87} C_VEL
LIN {X 0,Y 438.201,Z 619.605,A -85,B 0,C 180,E1 -8925.822,E2 -8925.822} C_VEL
LIN {X 0,Y 438.232,Z 618.199,A -85,B 0,C 180,E1 -8926.778,E2 -8926.778} C_VEL
LIN {X 0,Y 438.41,Z 615.191,A -85,B 0,C 180,E1 -8928.215,E2 -8928.215} C_VEL
LIN {X 0,Y 438.597,Z 611.044,A -85,B 0,C 180,E1 -8929.663,E2 -8929.663} C_VEL
LIN {X 0,Y 438.92,Z 604.546,A -85,B 0,C 180,E1 -8931.362,E2 -8931.362} C_VEL
LIN {X 0,Y 439.372,Z 597.385,A -85,B 0,C 180,E1 -8932.823,E2 -8932.823} C_VEL
LIN {X 0,Y 439.952,Z 588.962,A -85,B 0,C 180,E1 -8934.189,E2 -8934.189} C_VEL
LIN {X 0,Y 440.586,Z 578.812,A -85,B 0,C 180,E1 -8935.511,E2 -8935.511} C_VEL
LIN {X 0,Y 441.207,Z 569.533,A -85,B 0,C 180,E1 -8936.487,E2 -8936.487} C_VEL
LIN {X 0,Y 441.89,Z 559.149,A -85,B 0,C 180,E1 -8937.375,E2 -8937.375} C_VEL
LIN {X 0,Y 442.463,Z 547.952,A -85,B 0,C 180,E1 -8938.134,E2 -8938.134} C_VEL
LIN {X 0,Y 443.122,Z 534.837,A -85,B 0,C 180,E1 -8938.799,E2 -8938.799} C_VEL
LIN {X 0,Y 443.504,Z 522.296,A -85,B 0,C 180,E1 -8939.244,E2 -8939.244} C_VEL
LIN {X 0,Y 443.794,Z 506.6,A -85,B 0,C 180,E1 -8939.563,E2 -8939.563} C_VEL
LIN {X 0,Y 444.522,Z 429.048,A -85,B 0,C 180,E1 -8940.84,E2 -8940.84} C_VEL
LIN {X 0,Y 440.938,Z 410.776,A -85,B 0,C 180,E1 -8941.351,E2 -8941.351} C_VEL
LIN {X 0,Y 440.896,Z 409.741,A -85,B 0,C 180,E1 -8941.495,E2 -8941.495} C_VEL
LIN {X 0,Y 441.643,Z 397.54,A -85,B 0,C 180,E1 -8944.158,E2 -8944.158} C_VEL
LIN {X 0,Y 441.125,Z 392.689,A -85,B 0,C 180,E1 -8945.287,E2 -8945.287} C_VEL
LIN {X 0,Y 439.398,Z 384.299,A -85,B 0,C 180,E1 -8947.389,E2 -8947.389} C_VEL
LIN {X 0,Y 439.425,Z 384.25,A -85,B 0,C 180,E1 -8949.853,E2 -8949.853} C_VEL
LIN {X 0,Y 439.399,Z 384.252,A -85,B 0,C 180,E1 -8952.629,E2 -8952.629} C_VEL
LIN {X 0,Y 439.398,Z 384.25,A -85,B 0,C 180,E1 -8956.033,E2 -8956.033} C_VEL
LIN {X 0,Y 439.395,Z 384.252,A -85,B 0,C 180,E1 -8959.021,E2 -8959.021} C_VEL
LIN {X 0,Y 439.387,Z 384.249,A -85,B 0,C 180,E1 -8961.604,E2 -8961.604} C_VEL
LIN {X 0,Y 439.394,Z 384.247,A -85,B 0,C 180,E1 -8964.844,E2 -8964.844} C_VEL
LIN {X 0,Y 439.383,Z 384.251,A -85,B 0,C 180,E1 -8968.14,E2 -8968.14} C_VEL
LIN {X 0,Y 439.417,Z 384.245,A -85,B 0,C 180,E1 -8971.327,E2 -8971.327} C_VEL
LIN {X 0,Y 439.398,Z 384.25,A -85,B 0,C 180,E1 -8974.415,E2 -8974.415} C_VEL
LIN {X 0,Y 439.366,Z 384.251,A -85,B 0,C 180,E1 -8977.425,E2 -8977.425} C_VEL
LIN {X 0,Y 439.433,Z 384.248,A -85,B 0,C 180,E1 -8980.662,E2 -8980.662} C_VEL
LIN {X 0,Y 439.453,Z 384.242,A -85,B 0,C 180,E1 -8984.224,E2 -8984.224} C_VEL
LIN {X 0,Y 439.499,Z 384.236,A -85,B 0,C 180,E1 -8988.002,E2 -8988.002} C_VEL
LIN {X 0,Y 439.539,Z 384.231,A -85,B 0,C 180,E1 -8991.726,E2 -8991.726} C_VEL
LIN {X 0,Y 439.615,Z 384.22,A -85,B 0,C 180,E1 -8994.496,E2 -8994.496} C_VEL
LIN {X 0,Y 439.628,Z 384.219,A -85,B 0,C 180,E1 -8998.168,E2 -8998.168} C_VEL
LIN {X 0,Y 439.755,Z 384.201,A -85,B 0,C 180,E1 -9000,E2 -9000} C_VEL
LIN {X 0,Y 439.649,Z 384.22,A -85,B 0,C 180,E1 -9002.749,E2 -9002.749} C_VEL
LIN {X 0,Y 439.611,Z 384.225,A -85,B 0,C 180,E1 -9006.425,E2 -9006.425} C_VEL
LIN {X 0,Y 439.493,Z 384.236,A -85,B 0,C 180,E1 -9009.202,E2 -9009.202} C_VEL
LIN {X 0,Y 439.495,Z 384.237,A -85,B 0,C 180,E1 -9012.727,E2 -9012.727} C_VEL
LIN {X 0,Y 439.439,Z 384.246,A -85,B 0,C 180,E1 -9016.349,E2 -9016.349} C_VEL
LIN {X 0,Y 439.395,Z 384.247,A -85,B 0,C 180,E1 -9019.627,E2 -9019.627} C_VEL
LIN {X 0,Y 439.359,Z 384.254,A -85,B 0,C 180,E1 -9022.576,E2 -9022.576} C_VEL
LIN {X 0,Y 439.398,Z 384.247,A -85,B 0,C 180,E1 -9025.585,E2 -9025.585} C_VEL
LIN {X 0,Y 439.41,Z 384.254,A -85,B 0,C 180,E1 -9028.674,E2 -9028.674} C_VEL
LIN {X 0,Y 439.364,Z 384.253,A -85,B 0,C 180,E1 -9032.031,E2 -9032.031} C_VEL
LIN {X 0,Y 439.39,Z 384.25,A -85,B 0,C 180,E1 -9035.342,E2 -9035.342} C_VEL
LIN {X 0,Y 439.393,Z 384.255,A -85,B 0,C 180,E1 -9038.594,E2 -9038.594} C_VEL
LIN {X 0,Y 439.4,Z 384.237,A -85,B 0,C 180,E1 -9041.26,E2 -9041.26} C_VEL
LIN {X 0,Y 439.405,Z 384.249,A -85,B 0,C 180,E1 -9044.729,E2 -9044.729} C_VEL
LIN {X 0,Y 439.394,Z 384.249,A -85,B 0,C 180,E1 -9047.797,E2 -9047.797} C_VEL
LIN {X 0,Y 439.427,Z 384.243,A -85,B 0,C 180,E1 -9050.229,E2 -9050.229} C_VEL
LIN {X 0,Y 439.375,Z 384.248,A -85,B 0,C 180,E1 -9053.714,E2 -9053.714} C_VEL
LIN {X 0,Y 439.371,Z 384.256,A -85,B 0,C 180,E1 -9057.055,E2 -9057.055} C_VEL
LIN {X 0,Y 439.382,Z 384.253,A -85,B 0,C 180,E1 -9060.275,E2 -9060.275} C_VEL
LIN {X 0,Y 439.43,Z 384.248,A -85,B 0,C 180,E1 -9063.397,E2 -9063.397} C_VEL
LIN {X 0,Y 439.472,Z 384.401,A -85,B 0,C 180,E1 -9063.81,E2 -9063.81} C_VEL
LIN {X 0,Y 441.683,Z 395.29,A -85,B 0,C 180,E1 -9066.312,E2 -9066.312} C_VEL
LIN {X 0,Y 442.115,Z 399.487,A -85,B 0,C 180,E1 -9067.219,E2 -9067.219} C_VEL
LIN {X 0,Y 440.96,Z 417.827,A -85,B 0,C 180,E1 -9070.93,E2 -9070.93} C_VEL
LIN {X 0,Y 440.758,Z 421.789,A -85,B 0,C 180,E1 -9071.675,E2 -9071.675} C_VEL
LIN {X 0,Y 443.823,Z 439.101,A -85,B 0,C 180,E1 -9072.146,E2 -9072.146} C_VEL
LIN {X 0,Y 444.487,Z 444.367,A -85,B 0,C 180,E1 -9072.266,E2 -9072.266} C_VEL
LIN {X 0,Y 443.541,Z 530.016,A -85,B 0,C 180,E1 -9073.695,E2 -9073.695} C_VEL
LIN {X 0,Y 443.106,Z 543.78,A -85,B 0,C 180,E1 -9074.122,E2 -9074.122} C_VEL
LIN {X 0,Y 442.571,Z 556.143,A -85,B 0,C 180,E1 -9074.693,E2 -9074.693} C_VEL
LIN {X 0,Y 441.949,Z 567.198,A -85,B 0,C 180,E1 -9075.378,E2 -9075.378} C_VEL
LIN {X 0,Y 441.21,Z 579.1,A -85,B 0,C 180,E1 -9076.329,E2 -9076.329} C_VEL
LIN {X 0,Y 440.603,Z 589.107,A -85,B 0,C 180,E1 -9077.331,E2 -9077.331} C_VEL
LIN {X 0,Y 439.958,Z 598.47,A -85,B 0,C 180,E1 -9078.482,E2 -9078.482} C_VEL
LIN {X 0,Y 439.386,Z 607.513,A -85,B 0,C 180,E1 -9079.867,E2 -9079.867} C_VEL
LIN {X 0,Y 438.96,Z 614.811,A -85,B 0,C 180,E1 -9081.252,E2 -9081.252} C_VEL
LIN {X 0,Y 438.62,Z 620.67,A -85,B 0,C 180,E1 -9082.636,E2 -9082.636} C_VEL
LIN {X 0,Y 438.418,Z 625.056,A -85,B 0,C 180,E1 -9083.942,E2 -9083.942} C_VEL
LIN {X 0,Y 438.346,Z 628.823,A -85,B 0,C 180,E1 -9085.402,E2 -9085.402} C_VEL
LIN {X 0,Y 438.26,Z 630.623,A -85,B 0,C 180,E1 -9086.323,E2 -9086.323} C_VEL
LIN {X 0,Y 438.294,Z 631.982,A -85,B 0,C 180,E1 -9087.243,E2 -9087.243} C_VEL
LIN {X 0,Y 438.273,Z 632.948,A -85,B 0,C 180,E1 -9088.162,E2 -9088.162} C_VEL
LIN {X 0,Y 438.23,Z 633.528,A -85,B 0,C 180,E1 -9089.081,E2 -9089.081} C_VEL
LIN {X 0,Y 438.228,Z 633.696,A -85,B 0,C 180,E1 -9090,E2 -9090} C_VEL
LIN {X 0,Y 438.273,Z 632.815,A -85,B 0,C 180,E1 -9091.838,E2 -9091.838} C_VEL
LIN {X 0,Y 438.294,Z 631.794,A -85,B 0,C 180,E1 -9092.757,E2 -9092.757} C_VEL
LIN {X 0,Y 438.26,Z 630.347,A -85,B 0,C 180,E1 -9093.678,E2 -9093.678} C_VEL
LIN {X 0,Y 438.4,Z 627.363,A -85,B 0,C 180,E1 -9095.058,E2 -9095.058} C_VEL
LIN {X 0,Y 438.466,Z 623.321,A -85,B 0,C 180,E1 -9096.442,E2 -9096.442} C_VEL
LIN {X 0,Y 438.737,Z 617.1,A -85,B 0,C 180,E1 -9098.057,E2 -9098.057} C_VEL
LIN {X 0,Y 439.111,Z 610.315,A -85,B 0,C 180,E1 -9099.442,E2 -9099.442} C_VEL
LIN {X 0,Y 439.564,Z 601.872,A -85,B 0,C 180,E1 -9100.828,E2 -9100.828} C_VEL
LIN {X 0,Y 440.119,Z 593.161,A -85,B 0,C 180,E1 -9101.981,E2 -9101.981} C_VEL
LIN {X 0,Y 440.744,Z 582.177,A -85,B 0,C 180,E1 -9103.158,E2 -9103.158} C_VEL
LIN {X 0,Y 441.321,Z 571.737,A -85,B 0,C 180,E1 -9104.055,E2 -9104.055} C_VEL
LIN {X 0,Y 441.902,Z 559.756,A -85,B 0,C 180,E1 -9104.86,E2 -9104.86} C_VEL
LIN {X 0,Y 442.453,Z 547.271,A -85,B 0,C 180,E1 -9105.489,E2 -9105.489} C_VEL
LIN {X 0,Y 442.944,Z 534.332,A -85,B 0,C 180,E1 -9105.943,E2 -9105.943} C_VEL
LIN {X 0,Y 443.113,Z 518.666,A -85,B 0,C 180,E1 -9106.262,E2 -9106.262} C_VEL
LIN {X 0,Y 443.749,Z 442.165,A -85,B 0,C 180,E1 -9107.504,E2 -9107.504} C_VEL
LIN {X 0,Y 440.455,Z 421.853,A -85,B 0,C 180,E1 -9107.991,E2 -9107.991} C_VEL
LIN {X 0,Y 441.161,Z 407.565,A -85,B 0,C 180,E1 -9110.76,E2 -9110.76} C_VEL
LIN {X 0,Y 441.749,Z 397.938,A -85,B 0,C 180,E1 -9112.668,E2 -9112.668} C_VEL
LIN {X 0,Y 440.648,Z 390.418,A -85,B 0,C 180,E1 -9114.248,E2 -9114.248} C_VEL
LIN {X 0,Y 439.5,Z 384.332,A -85,B 0,C 180,E1 -9115.609,E2 -9115.609} C_VEL
LIN {X 0,Y 439.419,Z 384.249,A -85,B 0,C 180,E1 -9118.673,E2 -9118.673} C_VEL
LIN {X 0,Y 439.371,Z 384.253,A -85,B 0,C 180,E1 -9122.03,E2 -9122.03} C_VEL
LIN {X 0,Y 439.397,Z 384.254,A -85,B 0,C 180,E1 -9125.34,E2 -9125.34} C_VEL
LIN {X 0,Y 439.39,Z 384.25,A -85,B 0,C 180,E1 -9128.594,E2 -9128.594} C_VEL
LIN {X 0,Y 439.388,Z 384.254,A -85,B 0,C 180,E1 -9131.256,E2 -9131.256} C_VEL
LIN {X 0,Y 439.405,Z 384.249,A -85,B 0,C 180,E1 -9134.728,E2 -9134.728} C_VEL
LIN {X 0,Y 439.411,Z 384.249,A -85,B 0,C 180,E1 -9137.797,E2 -9137.797} C_VEL
LIN {X 0,Y 439.449,Z 384.243,A -85,B 0,C 180,E1 -9140.23,E2 -9140.23} C_VEL
LIN {X 0,Y 439.374,Z 384.254,A -85,B 0,C 180,E1 -9143.713,E2 -9143.713} C_VEL
LIN {X 0,Y 439.369,Z 384.256,A -85,B 0,C 180,E1 -9147.054,E2 -9147.054} C_VEL
LIN {X 0,Y 439.378,Z 384.253,A -85,B 0,C 180,E1 -9150.274,E2 -9150.274} C_VEL
LIN {X 0,Y 439.426,Z 384.249,A -85,B 0,C 180,E1 -9153.396,E2 -9153.396} C_VEL
LIN {X 0,Y 439.382,Z 384.252,A -85,B 0,C 180,E1 -9156.429,E2 -9156.429} C_VEL
LIN {X 0,Y 439.384,Z 384.254,A -85,B 0,C 180,E1 -9159.397,E2 -9159.397} C_VEL
LIN {X 0,Y 439.426,Z 384.247,A -85,B 0,C 180,E1 -9162.309,E2 -9162.309} C_VEL
LIN {X 0,Y 439.442,Z 384.248,A -85,B 0,C 180,E1 -9165.174,E2 -9165.174} C_VEL
LIN {X 0,Y 439.477,Z 384.242,A -85,B 0,C 180,E1 -9168.001,E2 -9168.001} C_VEL
LIN {X 0,Y 439.542,Z 384.234,A -85,B 0,C 180,E1 -9171.726,E2 -9171.726} C_VEL
LIN {X 0,Y 439.615,Z 384.224,A -85,B 0,C 180,E1 -9174.496,E2 -9174.496} C_VEL
LIN {X 0,Y 439.63,Z 384.222,A -85,B 0,C 180,E1 -9178.168,E2 -9178.168} C_VEL
LIN {X 0,Y 439.757,Z 384.207,A -85,B 0,C 180,E1 -9180,E2 -9180} C_VEL
LIN {X 0,Y 439.65,Z 384.221,A -85,B 0,C 180,E1 -9182.749,E2 -9182.749} C_VEL
LIN {X 0,Y 439.612,Z 384.224,A -85,B 0,C 180,E1 -9186.425,E2 -9186.425} C_VEL
LIN {X 0,Y 439.494,Z 384.24,A -85,B 0,C 180,E1 -9189.202,E2 -9189.202} C_VEL
LIN {X 0,Y 439.459,Z 384.244,A -85,B 0,C 180,E1 -9192.938,E2 -9192.938} C_VEL
LIN {X 0,Y 439.442,Z 384.245,A -85,B 0,C 180,E1 -9196.349,E2 -9196.349} C_VEL
LIN {X 0,Y 439.397,Z 384.253,A -85,B 0,C 180,E1 -9199.626,E2 -9199.626} C_VEL
LIN {X 0,Y 439.36,Z 384.257,A -85,B 0,C 180,E1 -9202.576,E2 -9202.576} C_VEL
LIN {X 0,Y 439.401,Z 384.253,A -85,B 0,C 180,E1 -9205.585,E2 -9205.585} C_VEL
LIN {X 0,Y 439.421,Z 384.249,A -85,B 0,C 180,E1 -9208.673,E2 -9208.673} C_VEL
LIN {X 0,Y 439.371,Z 384.254,A -85,B 0,C 180,E1 -9211.861,E2 -9211.861} C_VEL
LIN {X 0,Y 439.397,Z 384.253,A -85,B 0,C 180,E1 -9215.156,E2 -9215.156} C_VEL
LIN {X 0,Y 439.385,Z 384.253,A -85,B 0,C 180,E1 -9218.595,E2 -9218.595} C_VEL
LIN {X 0,Y 439.386,Z 384.255,A -85,B 0,C 180,E1 -9221.257,E2 -9221.257} C_VEL
LIN {X 0,Y 439.403,Z 384.25,A -85,B 0,C 180,E1 -9224.729,E2 -9224.729} C_VEL
LIN {X 0,Y 439.395,Z 384.251,A -85,B 0,C 180,E1 -9227.796,E2 -9227.796} C_VEL
LIN {X 0,Y 439.449,Z 384.244,A -85,B 0,C 180,E1 -9230.23,E2 -9230.23} C_VEL
LIN {X 0,Y 439.376,Z 384.253,A -85,B 0,C 180,E1 -9233.714,E2 -9233.714} C_VEL
LIN {X 0,Y 439.372,Z 384.257,A -85,B 0,C 180,E1 -9237.054,E2 -9237.054} C_VEL
LIN {X 0,Y 439.382,Z 384.251,A -85,B 0,C 180,E1 -9240.275,E2 -9240.275} C_VEL
LIN {X 0,Y 439.429,Z 384.248,A -85,B 0,C 180,E1 -9243.397,E2 -9243.397} C_VEL
LIN {X 0,Y 439.387,Z 384.251,A -85,B 0,C 180,E1 -9246.43,E2 -9246.43} C_VEL
LIN {X 0,Y 439.39,Z 384.252,A -85,B 0,C 180,E1 -9249.397,E2 -9249.397} C_VEL
LIN {X 0,Y 439.432,Z 384.245,A -85,B 0,C 180,E1 -9252.31,E2 -9252.31} C_VEL
LIN {X 0,Y 439.449,Z 384.248,A -85,B 0,C 180,E1 -9255.174,E2 -9255.174} C_VEL
LIN {X 0,Y 439.485,Z 384.242,A -85,B 0,C 180,E1 -9258.001,E2 -9258.001} C_VEL
LIN {X 0,Y 439.488,Z 384.359,A -85,B 0,C 180,E1 -9259.345,E2 -9259.345} C_VEL
LIN {X 0,Y 441.136,Z 393.139,A -85,B 0,C 180,E1 -9261.398,E2 -9261.398} C_VEL
LIN {X 0,Y 440.967,Z 401.139,A -85,B 0,C 180,E1 -9263.135,E2 -9263.135} C_VEL
LIN {X 0,Y 440.558,Z 409.758,A -85,B 0,C 180,E1 -9264.966,E2 -9264.966} C_VEL
LIN {X 0,Y 440.656,Z 411.192,A -85,B 0,C 180,E1 -9265.111,E2 -9265.111} C_VEL
LIN {X 0,Y 443.894,Z 429.704,A -85,B 0,C 180,E1 -9265.545,E2 -9265.545} C_VEL
LIN {X 0,Y 443.817,Z 438.209,A -85,B 0,C 180,E1 -9265.681,E2 -9265.681} C_VEL
LIN {X 0,Y 443.072,Z 444.052,A -85,B 0,C 180,E1 -9265.751,E2 -9265.751} C_VEL
LIN {X 0,Y 437.408,Z 463.043,A -85,B 0,C 180,E1 -9265.864,E2 -9265.864} C_VEL
LIN {X 0,Y 436.737,Z 468.884,A -85,B 0,C 180,E1 -9265.939,E2 -9265.939} C_VEL
LIN {X 0,Y 436.171,Z 517.888,A -85,B 0,C 180,E1 -9266.767,E2 -9266.767} C_VEL
LIN {X 0,Y 435.775,Z 530.948,A -85,B 0,C 180,E1 -9267.169,E2 -9267.169} C_VEL
LIN {X 0,Y 435.308,Z 543.519,A -85,B 0,C 180,E1 -9267.744,E2 -9267.744} C_VEL
LIN {X 0,Y 434.712,Z 555.53,A -85,B 0,C 180,E1 -9268.494,E2 -9268.494} C_VEL
LIN {X 0,Y 434.052,Z 566.975,A -85,B 0,C 180,E1 -9269.42,E2 -9269.42} C_VEL
LIN {X 0,Y 433.353,Z 577.311,A -85,B 0,C 180,E1 -9270.464,E2 -9270.464} C_VEL
LIN {X 0,Y 432.822,Z 586.589,A -85,B 0,C 180,E1 -9271.628,E2 -9271.628} C_VEL
LIN {X 0,Y 432.213,Z 595.596,A -85,B 0,C 180,E1 -9273.029,E2 -9273.029} C_VEL
LIN {X 0,Y 431.791,Z 602.861,A -85,B 0,C 180,E1 -9274.434,E2 -9274.434} C_VEL
LIN {X 0,Y 431.587,Z 608.994,A -85,B 0,C 180,E1 -9275.929,E2 -9275.929} C_VEL
LIN {X 0,Y 431.358,Z 613.904,A -85,B 0,C 180,E1 -9277.489,E2 -9277.489} C_VEL
LIN {X 0,Y 431.264,Z 616.237,A -85,B 0,C 180,E1 -9278.433,E2 -9278.433} C_VEL
LIN {X 0,Y 431.133,Z 618.143,A -85,B 0,C 180,E1 -9279.381,E2 -9279.381} C_VEL
LIN {X 0,Y 431.123,Z 619.571,A -85,B 0,C 180,E1 -9280.33,E2 -9280.33} C_VEL
LIN {X 0,Y 431.132,Z 621.093,A -85,B 0,C 180,E1 -9282.019,E2 -9282.019} C_VEL
LIN {X 0,Y 431.058,Z 621.418,A -85,B 0,C 180,E1 -9283.194,E2 -9283.194} C_VEL
LIN {X 0,Y 431.044,Z 621.177,A -85,B 0,C 180,E1 -9284.156,E2 -9284.156} C_VEL
LIN {X 0,Y 431.103,Z 619.728,A -85,B 0,C 180,E1 -9285.879,E2 -9285.879} C_VEL
LIN {X 0,Y 431.176,Z 617.953,A -85,B 0,C 180,E1 -9287.061,E2 -9287.061} C_VEL
LIN {X 0,Y 431.354,Z 614.799,A -85,B 0,C 180,E1 -9288.524,E2 -9288.524} C_VEL
LIN {X 0,Y 431.572,Z 610.485,A -85,B 0,C 180,E1 -9289.997,E2 -9289.997} C_VEL
LIN {X 0,Y 431.902,Z 604.871,A -85,B 0,C 180,E1 -9291.476,E2 -9291.476} C_VEL
LIN {X 0,Y 432.38,Z 597.759,A -85,B 0,C 180,E1 -9292.96,E2 -9292.96} C_VEL
LIN {X 0,Y 432.98,Z 589.411,A -85,B 0,C 180,E1 -9294.35,E2 -9294.35} C_VEL
LIN {X 0,Y 433.647,Z 579.35,A -85,B 0,C 180,E1 -9295.691,E2 -9295.691} C_VEL
LIN {X 0,Y 434.401,Z 568.925,A -85,B 0,C 180,E1 -9296.806,E2 -9296.806} C_VEL
LIN {X 0,Y 435.126,Z 558.509,A -85,B 0,C 180,E1 -9297.693,E2 -9297.693} C_VEL
LIN {X 0,Y 435.684,Z 547.964,A -85,B 0,C 180,E1 -9298.415,E2 -9298.415} C_VEL
LIN {X 0,Y 436.342,Z 535.543,A -85,B 0,C 180,E1 -9299.058,E2 -9299.058} C_VEL
LIN {X 0,Y 436.755,Z 522.953,A -85,B 0,C 180,E1 -9299.521,E2 -9299.521} C_VEL
LIN {X 0,Y 437.044,Z 508.838,A -85,B 0,C 180,E1 -9299.826,E2 -9299.826} C_VEL
LIN {X 0,Y 437.837,Z 429.83,A -85,B 0,C 180,E1 -9301.15,E2 -9301.15} C_VEL
LIN {X 0,Y 434.136,Z 411.461,A -85,B 0,C 180,E1 -9301.663,E2 -9301.663} C_VEL
LIN {X 0,Y 433.984,Z 410.273,A -85,B 0,C 180,E1 -9301.757,E2 -9301.757} C_VEL
LIN {X 0,Y 434.733,Z 398.037,A -85,B 0,C 180,E1 -9304.464,E2 -9304.464} C_VEL
LIN {X 0,Y 433.764,Z 392.115,A -85,B 0,C 180,E1 -9305.892,E2 -9305.892} C_VEL
LIN {X 0,Y 432.377,Z 385.173,A -85,B 0,C 180,E1 -9307.677,E2 -9307.677} C_VEL
LIN {X 0,Y 432.343,Z 385.133,A -85,B 0,C 180,E1 -9310.557,E2 -9310.557} C_VEL
LIN {X 0,Y 432.36,Z 385.127,A -85,B 0,C 180,E1 -9313.054,E2 -9313.054} C_VEL
LIN {X 0,Y 432.373,Z 385.126,A -85,B 0,C 180,E1 -9315.658,E2 -9315.658} C_VEL
LIN {X 0,Y 432.368,Z 385.121,A -85,B 0,C 180,E1 -9318.391,E2 -9318.391} C_VEL
LIN {X 0,Y 432.348,Z 385.125,A -85,B 0,C 180,E1 -9321.851,E2 -9321.851} C_VEL
LIN {X 0,Y 432.334,Z 385.124,A -85,B 0,C 180,E1 -9325.322,E2 -9325.322} C_VEL
LIN {X 0,Y 432.327,Z 385.133,A -85,B 0,C 180,E1 -9328.654,E2 -9328.654} C_VEL
LIN {X 0,Y 432.376,Z 385.122,A -85,B 0,C 180,E1 -9331.876,E2 -9331.876} C_VEL
LIN {X 0,Y 432.344,Z 385.13,A -85,B 0,C 180,E1 -9334.998,E2 -9334.998} C_VEL
LIN {X 0,Y 432.367,Z 385.12,A -85,B 0,C 180,E1 -9338.046,E2 -9338.046} C_VEL
LIN {X 0,Y 432.378,Z 385.124,A -85,B 0,C 180,E1 -9341.029,E2 -9341.029} C_VEL
LIN {X 0,Y 432.422,Z 385.117,A -85,B 0,C 180,E1 -9343.961,E2 -9343.961} C_VEL
LIN {X 0,Y 432.472,Z 385.111,A -85,B 0,C 180,E1 -9347.804,E2 -9347.804} C_VEL
LIN {X 0,Y 432.483,Z 385.111,A -85,B 0,C 180,E1 -9351.59,E2 -9351.59} C_VEL
LIN {X 0,Y 432.591,Z 385.094,A -85,B 0,C 180,E1 -9354.406,E2 -9354.406} C_VEL
LIN {X 0,Y 432.599,Z 385.094,A -85,B 0,C 180,E1 -9358.138,E2 -9358.138} C_VEL
LIN {X 0,Y 432.726,Z 385.076,A -85,B 0,C 180,E1 -9360,E2 -9360} C_VEL
LIN {X 0,Y 432.598,Z 385.097,A -85,B 0,C 180,E1 -9362.794,E2 -9362.794} C_VEL
LIN {X 0,Y 432.565,Z 385.103,A -85,B 0,C 180,E1 -9366.531,E2 -9366.531} C_VEL
LIN {X 0,Y 432.436,Z 385.114,A -85,B 0,C 180,E1 -9369.353,E2 -9369.353} C_VEL
LIN {X 0,Y 432.436,Z 385.115,A -85,B 0,C 180,E1 -9372.812,E2 -9372.812} C_VEL
LIN {X 0,Y 432.404,Z 385.124,A -85,B 0,C 180,E1 -9376.479,E2 -9376.479} C_VEL
LIN {X 0,Y 432.333,Z 385.128,A -85,B 0,C 180,E1 -9379.961,E2 -9379.961} C_VEL
LIN {X 0,Y 432.313,Z 385.131,A -85,B 0,C 180,E1 -9382.965,E2 -9382.965} C_VEL
LIN {X 0,Y 432.357,Z 385.125,A -85,B 0,C 180,E1 -9386.033,E2 -9386.033} C_VEL
LIN {X 0,Y 432.336,Z 385.129,A -85,B 0,C 180,E1 -9389.188,E2 -9389.188} C_VEL
LIN {X 0,Y 432.316,Z 385.135,A -85,B 0,C 180,E1 -9392.444,E2 -9392.444} C_VEL
LIN {X 0,Y 432.34,Z 385.128,A -85,B 0,C 180,E1 -9395.633,E2 -9395.633} C_VEL
LIN {X 0,Y 432.362,Z 385.125,A -85,B 0,C 180,E1 -9399.342,E2 -9399.342} C_VEL
LIN {X 0,Y 432.369,Z 385.112,A -85,B 0,C 180,E1 -9401.793,E2 -9401.793} C_VEL
LIN {X 0,Y 432.374,Z 385.129,A -85,B 0,C 180,E1 -9404.342,E2 -9404.342} C_VEL
LIN {X 0,Y 432.332,Z 385.132,A -85,B 0,C 180,E1 -9408.204,E2 -9408.204} C_VEL
LIN {X 0,Y 432.348,Z 385.129,A -85,B 0,C 180,E1 -9411.285,E2 -9411.285} C_VEL
LIN {X 0,Y 432.344,Z 385.129,A -85,B 0,C 180,E1 -9414.369,E2 -9414.369} C_VEL
LIN {X 0,Y 432.322,Z 385.133,A -85,B 0,C 180,E1 -9417.558,E2 -9417.558} C_VEL
LIN {X 0,Y 432.342,Z 385.133,A -85,B 0,C 180,E1 -9420.813,E2 -9420.813} C_VEL
LIN {X 0,Y 432.409,Z 385.225,A -85,B 0,C 180,E1 -9423.471,E2 -9423.471} C_VEL
LIN {X 0,Y 434.53,Z 395.437,A -85,B 0,C 180,E1 -9425.897,E2 -9425.897} C_VEL
LIN {X 0,Y 435.213,Z 400.367,A -85,B 0,C 180,E1 -9426.994,E2 -9426.994} C_VEL
LIN {X 0,Y 434.119,Z 416.724,A -85,B 0,C 180,E1 -9430.372,E2 -9430.372} C_VEL
LIN {X 0,Y 433.842,Z 421.503,A -85,B 0,C 180,E1 -9431.312,E2 -9431.312} C_VEL
LIN {X 0,Y 434.878,Z 426.98,A -85,B 0,C 180,E1 -9431.502,E2 -9431.502} C_VEL
LIN {X 0,Y 437.823,Z 444.423,A -85,B 0,C 180,E1 -9431.951,E2 -9431.951} C_VEL
LIN {X 0,Y 436.817,Z 530.11,A -85,B 0,C 180,E1 -9433.407,E2 -9433.407} C_VEL
LIN {X 0,Y 436.355,Z 543.793,A -85,B 0,C 180,E1 -9433.84,E2 -9433.84} C_VEL
LIN {X 0,Y 435.784,Z 555.57,A -85,B 0,C 180,E1 -9434.388,E2 -9434.388} C_VEL
LIN {X 0,Y 435.106,Z 567.527,A -85,B 0,C 180,E1 -9435.143,E2 -9435.143} C_VEL
LIN {X 0,Y 434.352,Z 578.954,A -85,B 0,C 180,E1 -9436.073,E2 -9436.073} C_VEL
LIN {X 0,Y 433.676,Z 589.278,A -85,B 0,C 180,E1 -9437.125,E2 -9437.125} C_VEL
LIN {X 0,Y 433.002,Z 598.577,A -85,B 0,C 180,E1 -9438.295,E2 -9438.295} C_VEL
LIN {X 0,Y 432.389,Z 607.584,A -85,B 0,C 180,E1 -9439.701,E2 -9439.701} C_VEL
LIN {X 0,Y 431.916,Z 614.853,A -85,B 0,C 180,E1 -9441.108,E2 -9441.108} C_VEL
LIN {X 0,Y 431.55,Z 620.685,A -85,B 0,C 180,E1 -9442.514,E2 -9442.514} C_VEL
LIN {X 0,Y 431.324,Z 625.445,A -85,B 0,C 180,E1 -9443.976,E2 -9443.976} C_VEL
LIN {X 0,Y 431.28,Z 628.79,A -85,B 0,C 180,E1 -9445.327,E2 -9445.327} C_VEL
LIN {X 0,Y 431.169,Z 630.568,A -85,B 0,C 180,E1 -9446.262,E2 -9446.262} C_VEL
LIN {X 0,Y 431.19,Z 631.916,A -85,B 0,C 180,E1 -9447.198,E2 -9447.198} C_VEL
LIN {X 0,Y 431.197,Z 632.872,A -85,B 0,C 180,E1 -9448.132,E2 -9448.132} C_VEL
LIN {X 0,Y 431.148,Z 633.442,A -85,B 0,C 180,E1 -9449.066,E2 -9449.066} C_VEL
LIN {X 0,Y 431.143,Z 633.59,A -85,B 0,C 180,E1 -9450,E2 -9450} C_VEL
LIN {X 0,Y 431.197,Z 632.69,A -85,B 0,C 180,E1 -9451.868,E2 -9451.868} C_VEL
LIN {X 0,Y 431.19,Z 631.659,A -85,B 0,C 180,E1 -9452.803,E2 -9452.803} C_VEL
LIN {X 0,Y 431.169,Z 630.191,A -85,B 0,C 180,E1 -9453.738,E2 -9453.738} C_VEL
LIN {X 0,Y 431.313,Z 627.186,A -85,B 0,C 180,E1 -9455.142,E2 -9455.142} C_VEL
LIN {X 0,Y 431.385,Z 623.119,A -85,B 0,C 180,E1 -9456.548,E2 -9456.548} C_VEL
LIN {X 0,Y 431.692,Z 616.866,A -85,B 0,C 180,E1 -9458.19,E2 -9458.19} C_VEL
LIN {X 0,Y 432.062,Z 610.05,A -85,B 0,C 180,E1 -9459.598,E2 -9459.598} C_VEL
LIN {X 0,Y 432.54,Z 601.554,A -85,B 0,C 180,E1 -9461.006,E2 -9461.006} C_VEL
LIN {X 0,Y 433.13,Z 592.799,A -85,B 0,C 180,E1 -9462.177,E2 -9462.177} C_VEL
LIN {X 0,Y 433.738,Z 582.731,A -85,B 0,C 180,E1 -9463.277,E2 -9463.277} C_VEL
LIN {X 0,Y 434.397,Z 571.235,A -85,B 0,C 180,E1 -9464.284,E2 -9464.284} C_VEL
LIN {X 0,Y 435.033,Z 559.124,A -85,B 0,C 180,E1 -9465.1,E2 -9465.1} C_VEL
LIN {X 0,Y 435.594,Z 546.475,A -85,B 0,C 180,E1 -9465.739,E2 -9465.739} C_VEL
LIN {X 0,Y 436.081,Z 534.161,A -85,B 0,C 180,E1 -9466.171,E2 -9466.171} C_VEL
LIN {X 0,Y 436.26,Z 518.45,A -85,B 0,C 180,E1 -9466.495,E2 -9466.495} C_VEL
LIN {X 0,Y 436.935,Z 443.1,A -85,B 0,C 180,E1 -9467.737,E2 -9467.737} C_VEL
LIN {X 0,Y 433.494,Z 421.812,A -85,B 0,C 180,E1 -9468.252,E2 -9468.252} C_VEL
LIN {X 0,Y 434.181,Z 408.499,A -85,B 0,C 180,E1 -9470.861,E2 -9470.861} C_VEL
LIN {X 0,Y 434.727,Z 397.641,A -85,B 0,C 180,E1 -9473.056,E2 -9473.056} C_VEL
LIN {X 0,Y 432.452,Z 385.216,A -85,B 0,C 180,E1 -9475.8,E2 -9475.8} C_VEL
LIN {X 0,Y 432.344,Z 385.133,A -85,B 0,C 180,E1 -9479.187,E2 -9479.187} C_VEL
LIN {X 0,Y 432.324,Z 385.129,A -85,B 0,C 180,E1 -9482.442,E2 -9482.442} C_VEL
LIN {X 0,Y 432.346,Z 385.132,A -85,B 0,C 180,E1 -9485.632,E2 -9485.632} C_VEL
LIN {X 0,Y 432.352,Z 385.126,A -85,B 0,C 180,E1 -9488.716,E2 -9488.716} C_VEL
LIN {X 0,Y 432.334,Z 385.131,A -85,B 0,C 180,E1 -9491.796,E2 -9491.796} C_VEL
LIN {X 0,Y 432.377,Z 385.127,A -85,B 0,C 180,E1 -9495.658,E2 -9495.658} C_VEL
LIN {X 0,Y 432.371,Z 385.125,A -85,B 0,C 180,E1 -9498.391,E2 -9498.391} C_VEL
LIN {X 0,Y 432.351,Z 385.128,A -85,B 0,C 180,E1 -9501.851,E2 -9501.851} C_VEL
LIN {X 0,Y 432.338,Z 385.134,A -85,B 0,C 180,E1 -9505.323,E2 -9505.323} C_VEL
LIN {X 0,Y 432.318,Z 385.132,A -85,B 0,C 180,E1 -9508.653,E2 -9508.653} C_VEL
LIN {X 0,Y 432.379,Z 385.125,A -85,B 0,C 180,E1 -9511.876,E2 -9511.876} C_VEL
LIN {X 0,Y 432.347,Z 385.131,A -85,B 0,C 180,E1 -9514.998,E2 -9514.998} C_VEL
LIN {X 0,Y 432.352,Z 385.129,A -85,B 0,C 180,E1 -9518.045,E2 -9518.045} C_VEL
LIN {X 0,Y 432.381,Z 385.128,A -85,B 0,C 180,E1 -9521.029,E2 -9521.029} C_VEL
LIN {X 0,Y 432.425,Z 385.12,A -85,B 0,C 180,E1 -9523.961,E2 -9523.961} C_VEL
LIN {X 0,Y 432.453,Z 385.117,A -85,B 0,C 180,E1 -9527.803,E2 -9527.803} C_VEL
LIN {X 0,Y 432.486,Z 385.113,A -85,B 0,C 180,E1 -9531.59,E2 -9531.59} C_VEL
LIN {X 0,Y 432.591,Z 385.098,A -85,B 0,C 180,E1 -9534.406,E2 -9534.406} C_VEL
LIN {X 0,Y 432.6,Z 385.098,A -85,B 0,C 180,E1 -9538.138,E2 -9538.138} C_VEL
LIN {X 0,Y 432.727,Z 385.082,A -85,B 0,C 180,E1 -9540,E2 -9540} C_VEL
LIN {X 0,Y 432.6,Z 385.1,A -85,B 0,C 180,E1 -9542.794,E2 -9542.794} C_VEL
LIN {X 0,Y 432.567,Z 385.102,A -85,B 0,C 180,E1 -9546.53,E2 -9546.53} C_VEL
LIN {X 0,Y 432.437,Z 385.119,A -85,B 0,C 180,E1 -9549.353,E2 -9549.353} C_VEL
LIN {X 0,Y 432.425,Z 385.121,A -85,B 0,C 180,E1 -9552.803,E2 -9552.803} C_VEL
LIN {X 0,Y 432.407,Z 385.122,A -85,B 0,C 180,E1 -9556.479,E2 -9556.479} C_VEL
LIN {X 0,Y 432.333,Z 385.131,A -85,B 0,C 180,E1 -9559.961,E2 -9559.961} C_VEL
LIN {X 0,Y 432.314,Z 385.134,A -85,B 0,C 180,E1 -9562.964,E2 -9562.964} C_VEL
LIN {X 0,Y 432.36,Z 385.127,A -85,B 0,C 180,E1 -9566.033,E2 -9566.033} C_VEL
LIN {X 0,Y 432.348,Z 385.131,A -85,B 0,C 180,E1 -9569.187,E2 -9569.187} C_VEL
LIN {X 0,Y 432.322,Z 385.132,A -85,B 0,C 180,E1 -9572.294,E2 -9572.294} C_VEL
LIN {X 0,Y 432.337,Z 385.131,A -85,B 0,C 180,E1 -9574.677,E2 -9574.677} C_VEL
LIN {X 0,Y 432.343,Z 385.129,A -85,B 0,C 180,E1 -9578.149,E2 -9578.149} C_VEL
LIN {X 0,Y 432.331,Z 385.132,A -85,B 0,C 180,E1 -9581.603,E2 -9581.603} C_VEL
LIN {X 0,Y 432.338,Z 385.13,A -85,B 0,C 180,E1 -9584.347,E2 -9584.347} C_VEL
LIN {X 0,Y 432.318,Z 385.134,A -85,B 0,C 180,E1 -9587.016,E2 -9587.016} C_VEL
LIN {X 0,Y 432.354,Z 385.127,A -85,B 0,C 180,E1 -9589.818,E2 -9589.818} C_VEL
LIN {X 0,Y 432.316,Z 385.135,A -85,B 0,C 180,E1 -9593.024,E2 -9593.024} C_VEL
LIN {X 0,Y 432.359,Z 385.126,A -85,B 0,C 180,E1 -9595.997,E2 -9595.997} C_VEL
LIN {X 0,Y 432.347,Z 385.129,A -85,B 0,C 180,E1 -9599.49,E2 -9599.49} C_VEL
LIN {X 0,Y 432.391,Z 385.126,A -85,B 0,C 180,E1 -9602.929,E2 -9602.929} C_VEL
LIN {X 0,Y 432.372,Z 385.124,A -85,B 0,C 180,E1 -9606.024,E2 -9606.024} C_VEL
LIN {X 0,Y 432.351,Z 385.133,A -85,B 0,C 180,E1 -9609.046,E2 -9609.046} C_VEL
LIN {X 0,Y 432.379,Z 385.123,A -85,B 0,C 180,E1 -9612.011,E2 -9612.011} C_VEL
LIN {X 0,Y 432.397,Z 385.127,A -85,B 0,C 180,E1 -9614.927,E2 -9614.927} C_VEL
LIN {X 0,Y 432.461,Z 385.117,A -85,B 0,C 180,E1 -9617.804,E2 -9617.804} C_VEL
LIN {X 0,Y 432.456,Z 385.247,A -85,B 0,C 180,E1 -9619.169,E2 -9619.169} C_VEL
LIN {X 0,Y 434.145,Z 394.228,A -85,B 0,C 180,E1 -9621.297,E2 -9621.297} C_VEL
LIN {X 0,Y 433.982,Z 402.078,A -85,B 0,C 180,E1 -9623.024,E2 -9623.024} C_VEL
LIN {X 0,Y 433.525,Z 409.618,A -85,B 0,C 180,E1 -9624.654,E2 -9624.654} C_VEL
LIN {X 0,Y 433.617,Z 410.693,A -85,B 0,C 180,E1 -9624.821,E2 -9624.821} C_VEL
LIN {X 0,Y 437.063,Z 430.153,A -85,B 0,C 180,E1 -9625.301,E2 -9625.301} C_VEL
LIN {X 0,Y 436.737,Z 468.884,A -85,B 0,C 180,E1 -9625.939,E2 -9625.939} C_VEL
LIN {X 0,Y 436.03,Z 474.729,A -85,B 0,C 180,E1 -9626.012,E2 -9626.012} C_VEL
LIN {X 0,Y 430.205,Z 493.693,A -85,B 0,C 180,E1 -9626.129,E2 -9626.129} C_VEL
LIN {X 0,Y 429.559,Z 499.535,A -85,B 0,C 180,E1 -9626.206,E2 -9626.206} C_VEL
LIN {X 0,Y 429.277,Z 519.163,A -85,B 0,C 180,E1 -9626.568,E2 -9626.568} C_VEL
LIN {X 0,Y 428.854,Z 532.592,A -85,B 0,C 180,E1 -9627.006,E2 -9627.006} C_VEL
LIN {X 0,Y 428.351,Z 544.726,A -85,B 0,C 180,E1 -9627.59,E2 -9627.59} C_VEL
LIN {X 0,Y 427.732,Z 556.459,A -85,B 0,C 180,E1 -9628.352,E2 -9628.352} C_VEL
LIN {X 0,Y 427.078,Z 567.754,A -85,B 0,C 180,E1 -9629.293,E2 -9629.293} C_VEL
LIN {X 0,Y 426.329,Z 577.978,A -85,B 0,C 180,E1 -9630.354,E2 -9630.354} C_VEL
LIN {X 0,Y 425.735,Z 587.947,A -85,B 0,C 180,E1 -9631.655,E2 -9631.655} C_VEL
LIN {X 0,Y 425.105,Z 596.753,A -85,B 0,C 180,E1 -9633.08,E2 -9633.08} C_VEL
LIN {X 0,Y 424.647,Z 603.807,A -85,B 0,C 180,E1 -9634.509,E2 -9634.509} C_VEL
LIN {X 0,Y 424.528,Z 608.581,A -85,B 0,C 180,E1 -9635.7,E2 -9635.7} C_VEL
LIN {X 0,Y 424.319,Z 613.22,A -85,B 0,C 180,E1 -9637.135,E2 -9637.135} C_VEL
LIN {X 0,Y 424.149,Z 616.759,A -85,B 0,C 180,E1 -9638.576,E2 -9638.576} C_VEL
LIN {X 0,Y 424.025,Z 618.547,A -85,B 0,C 180,E1 -9639.54,E2 -9639.54} C_VEL
LIN {X 0,Y 424.036,Z 619.895,A -85,B 0,C 180,E1 -9640.504,E2 -9640.504} C_VEL
LIN {X 0,Y 424.059,Z 621.222,A -85,B 0,C 180,E1 -9642.091,E2 -9642.091} C_VEL
LIN {X 0,Y 423.954,Z 621.489,A -85,B 0,C 180,E1 -9643.419,E2 -9643.419} C_VEL
LIN {X 0,Y 423.946,Z 621.181,A -85,B 0,C 180,E1 -9644.398,E2 -9644.398} C_VEL
LIN {X 0,Y 424.021,Z 619.797,A -85,B 0,C 180,E1 -9645.986,E2 -9645.986} C_VEL
LIN {X 0,Y 424.193,Z 616.732,A -85,B 0,C 180,E1 -9647.848,E2 -9647.848} C_VEL
LIN {X 0,Y 424.384,Z 613.055,A -85,B 0,C 180,E1 -9649.342,E2 -9649.342} C_VEL
LIN {X 0,Y 424.667,Z 608.159,A -85,B 0,C 180,E1 -9650.843,E2 -9650.843} C_VEL
LIN {X 0,Y 425.129,Z 601.885,A -85,B 0,C 180,E1 -9652.347,E2 -9652.347} C_VEL
LIN {X 0,Y 425.704,Z 593.983,A -85,B 0,C 180,E1 -9653.857,E2 -9653.857} C_VEL
LIN {X 0,Y 426.385,Z 584.95,A -85,B 0,C 180,E1 -9655.229,E2 -9655.229} C_VEL
LIN {X 0,Y 427.065,Z 575.624,A -85,B 0,C 180,E1 -9656.379,E2 -9656.379} C_VEL
LIN {X 0,Y 427.827,Z 565.606,A -85,B 0,C 180,E1 -9657.384,E2 -9657.384} C_VEL
LIN {X 0,Y 428.491,Z 554.684,A -85,B 0,C 180,E1 -9658.267,E2 -9658.267} C_VEL
LIN {X 0,Y 429.248,Z 542.585,A -85,B 0,C 180,E1 -9659.014,E2 -9659.014} C_VEL
LIN {X 0,Y 429.837,Z 529.223,A -85,B 0,C 180,E1 -9659.618,E2 -9659.618} C_VEL
LIN {X 0,Y 430.245,Z 516.778,A -85,B 0,C 180,E1 -9659.985,E2 -9659.985} C_VEL
LIN {X 0,Y 431.184,Z 430.502,A -85,B 0,C 180,E1 -9661.471,E2 -9661.471} C_VEL
LIN {X 0,Y 427.188,Z 411.199,A -85,B 0,C 180,E1 -9662.038,E2 -9662.038} C_VEL
LIN {X 0,Y 427.127,Z 410.094,A -85,B 0,C 180,E1 -9662.171,E2 -9662.171} C_VEL
LIN {X 0,Y 427.808,Z 400.365,A -85,B 0,C 180,E1 -9664.36,E2 -9664.36} C_VEL
LIN {X 0,Y 427.327,Z 395.914,A -85,B 0,C 180,E1 -9665.431,E2 -9665.431} C_VEL
LIN {X 0,Y 425.346,Z 386.192,A -85,B 0,C 180,E1 -9667.911,E2 -9667.911} C_VEL
LIN {X 0,Y 425.306,Z 386.007,A -85,B 0,C 180,E1 -9671.374,E2 -9671.374} C_VEL
LIN {X 0,Y 425.318,Z 386.006,A -85,B 0,C 180,E1 -9674.721,E2 -9674.721} C_VEL
LIN {X 0,Y 425.338,Z 385.995,A -85,B 0,C 180,E1 -9678.033,E2 -9678.033} C_VEL
LIN {X 0,Y 425.319,Z 386,A -85,B 0,C 180,E1 -9681.104,E2 -9681.104} C_VEL
LIN {X 0,Y 425.294,Z 386.004,A -85,B 0,C 180,E1 -9684.664,E2 -9684.664} C_VEL
LIN {X 0,Y 425.267,Z 386.009,A -85,B 0,C 180,E1 -9688.073,E2 -9688.073} C_VEL
LIN {X 0,Y 425.33,Z 386,A -85,B 0,C 180,E1 -9691.368,E2 -9691.368} C_VEL
LIN {X 0,Y 425.288,Z 386.008,A -85,B 0,C 180,E1 -9694.554,E2 -9694.554} C_VEL
LIN {X 0,Y 425.311,Z 385.999,A -85,B 0,C 180,E1 -9697.72,E2 -9697.72} C_VEL
LIN {X 0,Y 425.357,Z 386.002,A -85,B 0,C 180,E1 -9700.704,E2 -9700.704} C_VEL
LIN {X 0,Y 425.379,Z 385.995,A -85,B 0,C 180,E1 -9703.688,E2 -9703.688} C_VEL
LIN {X 0,Y 425.421,Z 385.99,A -85,B 0,C 180,E1 -9707.599,E2 -9707.599} C_VEL
LIN {X 0,Y 425.434,Z 385.99,A -85,B 0,C 180,E1 -9711.45,E2 -9711.45} C_VEL
LIN {X 0,Y 425.548,Z 385.971,A -85,B 0,C 180,E1 -9714.313,E2 -9714.313} C_VEL
LIN {X 0,Y 425.568,Z 385.97,A -85,B 0,C 180,E1 -9718.107,E2 -9718.107} C_VEL
LIN {X 0,Y 425.695,Z 385.952,A -85,B 0,C 180,E1 -9720,E2 -9720} C_VEL
LIN {X 0,Y 425.55,Z 385.974,A -85,B 0,C 180,E1 -9722.84,E2 -9722.84} C_VEL
LIN {X 0,Y 425.523,Z 385.982,A -85,B 0,C 180,E1 -9726.639,E2 -9726.639} C_VEL
LIN {X 0,Y 425.395,Z 385.99,A -85,B 0,C 180,E1 -9729.51,E2 -9729.51} C_VEL
LIN {X 0,Y 425.395,Z 385.991,A -85,B 0,C 180,E1 -9732.91,E2 -9732.91} C_VEL
LIN {X 0,Y 425.353,Z 386.004,A -85,B 0,C 180,E1 -9736.605,E2 -9736.605} C_VEL
LIN {X 0,Y 425.321,Z 386.001,A -85,B 0,C 180,E1 -9739.636,E2 -9739.636} C_VEL
LIN {X 0,Y 425.3,Z 386.003,A -85,B 0,C 180,E1 -9743.366,E2 -9743.366} C_VEL
LIN {X 0,Y 425.341,Z 386,A -85,B 0,C 180,E1 -9746.845,E2 -9746.845} C_VEL
LIN {X 0,Y 425.284,Z 386.006,A -85,B 0,C 180,E1 -9749.72,E2 -9749.72} C_VEL
LIN {X 0,Y 425.276,Z 386.008,A -85,B 0,C 180,E1 -9753.049,E2 -9753.049} C_VEL
LIN {X 0,Y 425.279,Z 386.009,A -85,B 0,C 180,E1 -9755.93,E2 -9755.93} C_VEL
LIN {X 0,Y 425.307,Z 386.006,A -85,B 0,C 180,E1 -9759.047,E2 -9759.047} C_VEL
LIN {X 0,Y 425.327,Z 385.998,A -85,B 0,C 180,E1 -9762.647,E2 -9762.647} C_VEL
LIN {X 0,Y 425.264,Z 386.005,A -85,B 0,C 180,E1 -9766.046,E2 -9766.046} C_VEL
LIN {X 0,Y 425.294,Z 386.01,A -85,B 0,C 180,E1 -9768.625,E2 -9768.625} C_VEL
LIN {X 0,Y 425.31,Z 386.006,A -85,B 0,C 180,E1 -9771.104,E2 -9771.104} C_VEL
LIN {X 0,Y 425.299,Z 386.011,A -85,B 0,C 180,E1 -9774.665,E2 -9774.665} C_VEL
LIN {X 0,Y 425.264,Z 386.012,A -85,B 0,C 180,E1 -9778.074,E2 -9778.074} C_VEL
LIN {X 0,Y 425.331,Z 386.005,A -85,B 0,C 180,E1 -9781.369,E2 -9781.369} C_VEL
LIN {X 0,Y 425.372,Z 386.099,A -85,B 0,C 180,E1 -9783.15,E2 -9783.15} C_VEL
LIN {X 0,Y 427.232,Z 394.961,A -85,B 0,C 180,E1 -9785.317,E2 -9785.317} C_VEL
LIN {X 0,Y 428.307,Z 401.467,A -85,B 0,C 180,E1 -9786.809,E2 -9786.809} C_VEL
LIN {X 0,Y 427.34,Z 415.663,A -85,B 0,C 180,E1 -9789.797,E2 -9789.797} C_VEL
LIN {X 0,Y 427.014,Z 421.582,A -85,B 0,C 180,E1 -9790.975,E2 -9790.975} C_VEL
LIN {X 0,Y 430.236,Z 439.031,A -85,B 0,C 180,E1 -9791.48,E2 -9791.48} C_VEL
LIN {X 0,Y 431.143,Z 446.116,A -85,B 0,C 180,E1 -9791.651,E2 -9791.651} C_VEL
LIN {X 0,Y 430.124,Z 529.166,A -85,B 0,C 180,E1 -9793.08,E2 -9793.08} C_VEL
LIN {X 0,Y 429.676,Z 542.37,A -85,B 0,C 180,E1 -9793.49,E2 -9793.49} C_VEL
LIN {X 0,Y 429.061,Z 555.048,A -85,B 0,C 180,E1 -9794.076,E2 -9794.076} C_VEL
LIN {X 0,Y 428.329,Z 566.339,A -85,B 0,C 180,E1 -9794.781,E2 -9794.781} C_VEL
LIN {X 0,Y 427.589,Z 577.975,A -85,B 0,C 180,E1 -9795.727,E2 -9795.727} C_VEL
LIN {X 0,Y 426.833,Z 588.443,A -85,B 0,C 180,E1 -9796.794,E2 -9796.794} C_VEL
LIN {X 0,Y 426.238,Z 597.009,A -85,B 0,C 180,E1 -9797.865,E2 -9797.865} C_VEL
LIN {X 0,Y 425.556,Z 604.919,A -85,B 0,C 180,E1 -9799.052,E2 -9799.052} C_VEL
LIN {X 0,Y 425.032,Z 612.674,A -85,B 0,C 180,E1 -9800.483,E2 -9800.483} C_VEL
LIN {X 0,Y 424.594,Z 618.893,A -85,B 0,C 180,E1 -9801.912,E2 -9801.912} C_VEL
LIN {X 0,Y 424.296,Z 624.731,A -85,B 0,C 180,E1 -9803.637,E2 -9803.637} C_VEL
LIN {X 0,Y 424.213,Z 628.757,A -85,B 0,C 180,E1 -9805.249,E2 -9805.249} C_VEL
LIN {X 0,Y 424.083,Z 630.514,A -85,B 0,C 180,E1 -9806.199,E2 -9806.199} C_VEL
LIN {X 0,Y 424.121,Z 632.798,A -85,B 0,C 180,E1 -9808.101,E2 -9808.101} C_VEL
LIN {X 0,Y 424.069,Z 633.356,A -85,B 0,C 180,E1 -9809.051,E2 -9809.051} C_VEL
LIN {X 0,Y 424.062,Z 633.485,A -85,B 0,C 180,E1 -9810,E2 -9810} C_VEL
LIN {X 0,Y 424.122,Z 632.564,A -85,B 0,C 180,E1 -9811.899,E2 -9811.899} C_VEL
LIN {X 0,Y 424.087,Z 631.521,A -85,B 0,C 180,E1 -9812.85,E2 -9812.85} C_VEL
LIN {X 0,Y 424.083,Z 630.031,A -85,B 0,C 180,E1 -9813.801,E2 -9813.801} C_VEL
LIN {X 0,Y 424.226,Z 627.004,A -85,B 0,C 180,E1 -9815.228,E2 -9815.228} C_VEL
LIN {X 0,Y 424.308,Z 622.911,A -85,B 0,C 180,E1 -9816.658,E2 -9816.658} C_VEL
LIN {X 0,Y 424.629,Z 616.631,A -85,B 0,C 180,E1 -9818.327,E2 -9818.327} C_VEL
LIN {X 0,Y 425.026,Z 609.784,A -85,B 0,C 180,E1 -9819.758,E2 -9819.758} C_VEL
LIN {X 0,Y 425.536,Z 601.235,A -85,B 0,C 180,E1 -9821.19,E2 -9821.19} C_VEL
LIN {X 0,Y 426.149,Z 592.428,A -85,B 0,C 180,E1 -9822.38,E2 -9822.38} C_VEL
LIN {X 0,Y 426.81,Z 581.699,A -85,B 0,C 180,E1 -9823.558,E2 -9823.558} C_VEL
LIN {X 0,Y 427.468,Z 570.675,A -85,B 0,C 180,E1 -9824.52,E2 -9824.52} C_VEL
LIN {X 0,Y 428.12,Z 558.424,A -85,B 0,C 180,E1 -9825.349,E2 -9825.349} C_VEL
LIN {X 0,Y 428.756,Z 545.578,A -85,B 0,C 180,E1 -9825.997,E2 -9825.997} C_VEL
LIN {X 0,Y 429.194,Z 532.657,A -85,B 0,C 180,E1 -9826.438,E2 -9826.438} C_VEL
LIN {X 0,Y 429.476,Z 514.359,A -85,B 0,C 180,E1 -9826.794,E2 -9826.794} C_VEL
LIN {X 0,Y 430.047,Z 443.684,A -85,B 0,C 180,E1 -9827.98,E2 -9827.98} C_VEL
LIN {X 0,Y 426.545,Z 421.673,A -85,B 0,C 180,E1 -9828.519,E2 -9828.519} C_VEL
LIN {X 0,Y 427.318,Z 406.971,A -85,B 0,C 180,E1 -9831.465,E2 -9831.465} C_VEL
LIN {X 0,Y 427.778,Z 399.16,A -85,B 0,C 180,E1 -9833.069,E2 -9833.069} C_VEL
LIN {X 0,Y 425.627,Z 387.273,A -85,B 0,C 180,E1 -9835.686,E2 -9835.686} C_VEL
LIN {X 0,Y 425.375,Z 386.034,A -85,B 0,C 180,E1 -9836.031,E2 -9836.031} C_VEL
LIN {X 0,Y 425.33,Z 386.005,A -85,B 0,C 180,E1 -9838.865,E2 -9838.865} C_VEL
LIN {X 0,Y 425.266,Z 386.011,A -85,B 0,C 180,E1 -9841.926,E2 -9841.926} C_VEL
LIN {X 0,Y 425.301,Z 386.009,A -85,B 0,C 180,E1 -9845.335,E2 -9845.335} C_VEL
LIN {X 0,Y 425.303,Z 386.006,A -85,B 0,C 180,E1 -9849.044,E2 -9849.044} C_VEL
LIN {X 0,Y 425.277,Z 386.008,A -85,B 0,C 180,E1 -9852.652,E2 -9852.652} C_VEL
LIN {X 0,Y 425.317,Z 386.004,A -85,B 0,C 180,E1 -9856.051,E2 -9856.051} C_VEL
LIN {X 0,Y 425.308,Z 386.004,A -85,B 0,C 180,E1 -9858.625,E2 -9858.625} C_VEL
LIN {X 0,Y 425.322,Z 386.006,A -85,B 0,C 180,E1 -9861.104,E2 -9861.104} C_VEL
LIN {X 0,Y 425.297,Z 386.006,A -85,B 0,C 180,E1 -9864.664,E2 -9864.664} C_VEL
LIN {X 0,Y 425.261,Z 386.012,A -85,B 0,C 180,E1 -9868.073,E2 -9868.073} C_VEL
LIN {X 0,Y 425.327,Z 386.006,A -85,B 0,C 180,E1 -9871.367,E2 -9871.367} C_VEL
LIN {X 0,Y 425.291,Z 386.007,A -85,B 0,C 180,E1 -9874.554,E2 -9874.554} C_VEL
LIN {X 0,Y 425.283,Z 386.01,A -85,B 0,C 180,E1 -9877.661,E2 -9877.661} C_VEL
LIN {X 0,Y 425.357,Z 386,A -85,B 0,C 180,E1 -9880.704,E2 -9880.704} C_VEL
LIN {X 0,Y 425.383,Z 385.997,A -85,B 0,C 180,E1 -9883.688,E2 -9883.688} C_VEL
LIN {X 0,Y 425.406,Z 385.995,A -85,B 0,C 180,E1 -9887.598,E2 -9887.598} C_VEL
LIN {X 0,Y 425.437,Z 385.991,A -85,B 0,C 180,E1 -9891.45,E2 -9891.45} C_VEL
LIN {X 0,Y 425.548,Z 385.975,A -85,B 0,C 180,E1 -9894.313,E2 -9894.313} C_VEL
LIN {X 0,Y 425.569,Z 385.973,A -85,B 0,C 180,E1 -9898.107,E2 -9898.107} C_VEL
LIN {X 0,Y 425.697,Z 385.958,A -85,B 0,C 180,E1 -9900,E2 -9900} C_VEL
LIN {X 0,Y 425.552,Z 385.978,A -85,B 0,C 180,E1 -9902.84,E2 -9902.84} C_VEL
LIN {X 0,Y 425.524,Z 385.98,A -85,B 0,C 180,E1 -9906.647,E2 -9906.647} C_VEL
LIN {X 0,Y 425.395,Z 385.997,A -85,B 0,C 180,E1 -9909.509,E2 -9909.509} C_VEL
LIN {X 0,Y 425.387,Z 385.998,A -85,B 0,C 180,E1 -9912.904,E2 -9912.904} C_VEL
LIN {X 0,Y 425.356,Z 386.001,A -85,B 0,C 180,E1 -9916.605,E2 -9916.605} C_VEL
LIN {X 0,Y 425.323,Z 386.006,A -85,B 0,C 180,E1 -9919.636,E2 -9919.636} C_VEL
LIN {X 0,Y 425.302,Z 386.009,A -85,B 0,C 180,E1 -9923.365,E2 -9923.365} C_VEL
LIN {X 0,Y 425.344,Z 386.003,A -85,B 0,C 180,E1 -9926.845,E2 -9926.845} C_VEL
LIN {X 0,Y 425.314,Z 386.006,A -85,B 0,C 180,E1 -9929.718,E2 -9929.718} C_VEL
LIN {X 0,Y 425.278,Z 386.011,A -85,B 0,C 180,E1 -9933.048,E2 -9933.048} C_VEL
LIN {X 0,Y 425.281,Z 386.009,A -85,B 0,C 180,E1 -9935.93,E2 -9935.93} C_VEL
LIN {X 0,Y 425.297,Z 386.009,A -85,B 0,C 180,E1 -9939.044,E2 -9939.044} C_VEL
LIN {X 0,Y 425.275,Z 386.01,A -85,B 0,C 180,E1 -9942.653,E2 -9942.653} C_VEL
LIN {X 0,Y 425.259,Z 386.011,A -85,B 0,C 180,E1 -9946.045,E2 -9946.045} C_VEL
LIN {X 0,Y 425.302,Z 386.007,A -85,B 0,C 180,E1 -9948.625,E2 -9948.625} C_VEL
LIN {X 0,Y 425.322,Z 386.007,A -85,B 0,C 180,E1 -9951.105,E2 -9951.105} C_VEL
LIN {X 0,Y 425.3,Z 386.007,A -85,B 0,C 180,E1 -9954.665,E2 -9954.665} C_VEL
LIN {X 0,Y 425.264,Z 386.01,A -85,B 0,C 180,E1 -9958.073,E2 -9958.073} C_VEL
LIN {X 0,Y 425.331,Z 386.004,A -85,B 0,C 180,E1 -9961.368,E2 -9961.368} C_VEL
LIN {X 0,Y 425.296,Z 386.007,A -85,B 0,C 180,E1 -9964.555,E2 -9964.555} C_VEL
LIN {X 0,Y 425.288,Z 386.007,A -85,B 0,C 180,E1 -9967.662,E2 -9967.662} C_VEL
LIN {X 0,Y 425.363,Z 386,A -85,B 0,C 180,E1 -9970.704,E2 -9970.704} C_VEL
LIN {X 0,Y 425.39,Z 385.993,A -85,B 0,C 180,E1 -9973.688,E2 -9973.688} C_VEL
LIN {X 0,Y 425.414,Z 385.994,A -85,B 0,C 180,E1 -9977.598,E2 -9977.598} C_VEL
LIN {X 0,Y 425.396,Z 386.133,A -85,B 0,C 180,E1 -9978.987,E2 -9978.987} C_VEL
LIN {X 0,Y 427.237,Z 396.584,A -85,B 0,C 180,E1 -9981.486,E2 -9981.486} C_VEL
LIN {X 0,Y 426.781,Z 404.078,A -85,B 0,C 180,E1 -9983.143,E2 -9983.143} C_VEL
LIN {X 0,Y 426.545,Z 410.587,A -85,B 0,C 180,E1 -9984.531,E2 -9984.531} C_VEL
LIN {X 0,Y 428.281,Z 420.148,A -85,B 0,C 180,E1 -9984.799,E2 -9984.799} C_VEL
LIN {X 0,Y 430.246,Z 431.073,A -85,B 0,C 180,E1 -9985.062,E2 -9985.062} C_VEL
LIN {X 0,Y 429.559,Z 499.535,A -85,B 0,C 180,E1 -9986.206,E2 -9986.206} C_VEL
LIN {X 0,Y 428.975,Z 505.37,A -85,B 0,C 180,E1 -9986.283,E2 -9986.283} C_VEL
LIN {X 0,Y 426.26,Z 514.855,A -85,B 0,C 180,E1 -9986.363,E2 -9986.363} C_VEL
LIN {X 0,Y 423.208,Z 524.24,A -85,B 0,C 180,E1 -9986.502,E2 -9986.502} C_VEL
LIN {X 0,Y 422.1,Z 529.926,A -85,B 0,C 180,E1 -9986.669,E2 -9986.669} C_VEL
LIN {X 0,Y 421.555,Z 542.65,A -85,B 0,C 180,E1 -9987.253,E2 -9987.253} C_VEL
LIN {X 0,Y 420.976,Z 554.143,A -85,B 0,C 180,E1 -9987.967,E2 -9987.967} C_VEL
LIN {X 0,Y 420.225,Z 565.94,A -85,B 0,C 180,E1 -9988.922,E2 -9988.922} C_VEL
LIN {X 0,Y 419.499,Z 576.486,A -85,B 0,C 180,E1 -9990,E2 -9990} C_VEL
LIN {X 0,Y 418.864,Z 585.996,A -85,B 0,C 180,E1 -9991.202,E2 -9991.202} C_VEL
LIN {X 0,Y 418.197,Z 595.163,A -85,B 0,C 180,E1 -9992.649,E2 -9992.649} C_VEL
LIN {X 0,Y 417.764,Z 602.538,A -85,B 0,C 180,E1 -9994.1,E2 -9994.1} C_VEL
LIN {X 0,Y 417.463,Z 607.56,A -85,B 0,C 180,E1 -9995.312,E2 -9995.312} C_VEL
LIN {X 0,Y 417.272,Z 612.432,A -85,B 0,C 180,E1 -9996.77,E2 -9996.77} C_VEL
LIN {X 0,Y 417.093,Z 616.193,A -85,B 0,C 180,E1 -9998.234,E2 -9998.234} C_VEL
LIN {X 0,Y 416.921,Z 618.929,A -85,B 0,C 180,E1 -9999.704,E2 -9999.704} C_VEL
LIN {X 0,Y 416.958,Z 620.213,A -85,B 0,C 180,E1 -10000.685,E2 -10000.685} C_VEL
LIN {X 0,Y 416.975,Z 621.346,A -85,B 0,C 180,E1 -10002.157,E2 -10002.157} C_VEL
LIN {X 0,Y 416.843,Z 621.559,A -85,B 0,C 180,E1 -10003.652,E2 -10003.652} C_VEL
LIN {X 0,Y 416.867,Z 621.188,A -85,B 0,C 180,E1 -10004.648,E2 -10004.648} C_VEL
LIN {X 0,Y 416.939,Z 619.872,A -85,B 0,C 180,E1 -10006.095,E2 -10006.095} C_VEL
LIN {X 0,Y 417.136,Z 616.414,A -85,B 0,C 180,E1 -10008.161,E2 -10008.161} C_VEL
LIN {X 0,Y 417.362,Z 612.593,A -85,B 0,C 180,E1 -10009.68,E2 -10009.68} C_VEL
LIN {X 0,Y 417.702,Z 607.542,A -85,B 0,C 180,E1 -10011.207,E2 -10011.207} C_VEL
LIN {X 0,Y 418.191,Z 601.094,A -85,B 0,C 180,E1 -10012.738,E2 -10012.738} C_VEL
LIN {X 0,Y 418.717,Z 594.423,A -85,B 0,C 180,E1 -10014.017,E2 -10014.017} C_VEL
LIN {X 0,Y 419.459,Z 585.366,A -85,B 0,C 180,E1 -10015.428,E2 -10015.428} C_VEL
LIN {X 0,Y 420.244,Z 575.134,A -85,B 0,C 180,E1 -10016.707,E2 -10016.707} C_VEL
